C09108=1015.374,-2.873,381.493,-24.167,21.529,-42.895
C09109=1015.372,-2.524,381.465,-24.168,21.529,-42.890
C09110=1015.370,-2.175,381.437,-24.169,21.528,-42.886
C09111=1015.368,-1.829,381.408,-24.169,21.528,-42.880
C09112=1015.365,-1.484,381.381,-24.170,21.527,-42.877
C09113=1015.363,-1.141,381.352,-24.170,21.527,-42.873
C09114=1015.360,-0.799,381.325,-24.171,21.526,-42.867
C09115=1015.359,-0.459,381.298,-24.172,21.526,-42.864
C09116=1015.357,-0.120,381.270,-24.172,21.526,-42.858
C09117=1015.353,0.217,381.242,-24.173,21.525,-42.855
C09118=1015.351,0.553,381.215,-24.173,21.525,-42.851
C09119=1015.350,0.887,381.188,-24.174,21.525,-42.846
C09120=1015.347,1.221,381.161,-24.175,21.524,-42.842
C09121=1015.344,1.555,381.134,-24.175,21.523,-42.838
C09122=1015.342,1.885,381.106,-24.176,21.523,-42.834
C09123=1015.340,2.198,381.082,-24.176,21.523,-42.831
C09124=1015.339,2.486,381.058,-24.177,21.522,-42.827
C09125=1015.336,2.755,381.036,-24.177,21.522,-42.823
C09126=1015.334,3.017,381.015,-24.178,21.522,-42.818
C09127=1015.333,3.286,380.993,-24.179,21.521,-42.814
C09128=1015.330,3.575,380.969,-24.179,21.521,-42.810
C09129=1015.328,3.889,380.943,-24.179,21.520,-42.807
C09130=1015.326,4.218,380.916,-24.180,21.521,-42.803
C09131=1015.323,4.550,380.890,-24.180,21.519,-42.799
C09132=1015.321,4.881,380.862,-24.181,21.519,-42.795
C09133=1015.318,5.211,380.836,-24.181,21.518,-42.792
C09134=1015.316,5.542,380.808,-24.182,21.519,-42.786
C09135=1015.314,5.872,380.782,-24.183,21.518,-42.783
C09136=1015.311,6.201,380.754,-24.183,21.518,-42.779
C09137=1015.308,6.530,380.728,-24.184,21.518,-42.774
C09138=1015.306,6.858,380.701,-24.185,21.517,-42.770
C09139=1015.303,7.186,380.674,-24.185,21.517,-42.766
C09140=1015.301,7.512,380.647,-24.186,21.516,-42.762
C09141=1015.298,7.834,380.620,-24.186,21.516,-42.759
C09142=1015.295,8.155,380.594,-24.186,21.515,-42.755
C09143=1015.294,8.473,380.568,-24.187,21.516,-42.750
C09144=1015.290,8.790,380.542,-24.188,21.515,-42.746
C09145=1015.288,9.105,380.517,-24.188,21.515,-42.742
C09146=1015.285,9.420,380.491,-24.189,21.514,-42.738
C09147=1015.283,9.735,380.465,-24.190,21.514,-42.733
C09148=1015.280,10.050,380.439,-24.190,21.514,-42.730
C09149=1015.278,10.367,380.413,-24.191,21.513,-42.726
C09150=1015.275,10.685,380.387,-24.191,21.513,-42.722
C09151=1015.272,11.006,380.361,-24.192,21.512,-42.718
C09152=1015.269,11.328,380.334,-24.192,21.512,-42.715
C09153=1015.267,11.652,380.307,-24.193,21.511,-42.711
C09154=1015.264,11.975,380.281,-24.193,21.511,-42.707
C09155=1015.261,12.298,380.254,-24.194,21.511,-42.702
C09156=1015.259,12.622,380.227,-24.194,21.510,-42.698
C09157=1015.255,12.945,380.201,-24.195,21.510,-42.694
C09158=1015.253,13.270,380.174,-24.195,21.509,-42.691
C09159=1015.250,13.593,380.148,-24.196,21.509,-42.687
C09160=1015.247,13.918,380.121,-24.197,21.509,-42.682
C09161=1015.244,14.242,380.094,-24.197,21.509,-42.678
C09162=1015.241,14.568,380.068,-24.198,21.508,-42.674
C09163=1015.238,14.893,380.041,-24.198,21.508,-42.670
C09164=1015.235,15.218,380.014,-24.199,21.507,-42.667
C09165=1015.233,15.545,379.987,-24.199,21.507,-42.663
C09166=1015.229,15.872,379.960,-24.200,21.507,-42.658
C09167=1015.227,16.199,379.933,-24.200,21.506,-42.654
C09168=1015.223,16.527,379.906,-24.201,21.506,-42.650
C09169=1015.220,16.856,379.878,-24.201,21.505,-42.646
C09170=1015.217,17.185,379.851,-24.202,21.505,-42.643
C09171=1015.214,17.516,379.824,-24.202,21.504,-42.639
C09172=1015.211,17.845,379.797,-24.203,21.504,-42.634
C09173=1015.208,18.175,379.770,-24.204,21.504,-42.630
C09174=1015.204,18.508,379.742,-24.204,21.503,-42.626
C09175=1015.202,18.839,379.715,-24.205,21.503,-42.622
C09176=1015.198,19.171,379.687,-24.205,21.502,-42.619
C09177=1015.195,19.519,379.658,-24.206,21.503,-42.613
C09178=1015.191,19.937,379.623,-24.207,21.502,-42.608
C09179=1015.188,20.173,379.604,-24.207,21.502,-42.604
C09180=1015.186,20.419,379.584,-24.207,21.502,-42.603
C09181=1015.183,20.668,379.563,-24.208,21.502,-42.601
C09182=1015.180,20.909,379.544,-24.208,21.502,-42.599
C09183=1015.179,21.136,379.524,-24.208,21.501,-42.597
C09184=1015.176,21.344,379.507,-24.209,21.501,-42.593
C09185=1015.172,21.701,379.478,-24.209,21.500,-42.588
C09186=1015.169,22.024,379.451,-24.210,21.501,-42.584
C09187=1015.166,22.319,379.426,-24.210,21.500,-42.582
C09188=1015.164,22.571,379.405,-24.210,21.499,-42.580
C09189=1015.159,22.981,379.371,-24.211,21.499,-42.573
C09190=1015.155,23.388,379.338,-24.212,21.498,-42.565
C09191=1015.153,23.641,379.316,-24.213,21.498,-42.562
C09192=1015.149,23.935,379.292,-24.213,21.498,-42.560
C09193=1015.146,24.262,379.265,-24.213,21.497,-42.558
C09194=1015.143,24.596,379.237,-24.214,21.497,-42.553
C09195=1015.139,24.930,379.209,-24.215,21.497,-42.549
C09196=1015.135,25.264,379.182,-24.215,21.496,-42.545
C09197=1015.132,25.598,379.155,-24.216,21.496,-42.541
C09198=1015.128,25.933,379.127,-24.216,21.495,-42.538
C09199=1015.124,26.266,379.098,-24.217,21.495,-42.534
C09200=1015.121,26.601,379.070,-24.217,21.494,-42.530
C09201=1015.117,26.935,379.043,-24.218,21.494,-42.525
C09202=1015.114,27.269,379.015,-24.219,21.495,-42.522
C09203=1015.110,27.604,378.987,-24.219,21.494,-42.518
C09204=1015.106,27.939,378.959,-24.220,21.494,-42.514
C09205=1015.102,28.273,378.932,-24.220,21.493,-42.510
C09206=1015.098,28.608,378.904,-24.221,21.493,-42.507
C09207=1015.095,28.942,378.876,-24.221,21.492,-42.503
C09208=1015.091,29.276,378.848,-24.222,21.493,-42.498
C09209=1015.087,29.611,378.820,-24.222,21.492,-42.494
C09210=1015.083,29.945,378.792,-24.223,21.492,-42.490
C09211=1015.079,30.280,378.764,-24.223,21.491,-42.486
C09212=1015.075,30.613,378.736,-24.224,21.491,-42.483
C09213=1015.071,30.948,378.708,-24.224,21.490,-42.479
C09214=1015.068,31.282,378.680,-24.225,21.490,-42.475
C09215=1015.063,31.617,378.652,-24.225,21.489,-42.471
C09216=1015.059,31.951,378.624,-24.226,21.489,-42.468
C09217=1015.055,32.286,378.597,-24.226,21.489,-42.464
C09218=1015.051,32.621,378.569,-24.227,21.489,-42.459
C09219=1015.048,32.955,378.541,-24.228,21.489,-42.455
C09220=1015.043,33.290,378.512,-24.228,21.488,-42.452
C09221=1015.039,33.624,378.484,-24.229,21.488,-42.448
C09222=1015.036,33.959,378.456,-24.229,21.487,-42.444
C09223=1015.031,34.294,378.428,-24.230,21.487,-42.440
C09224=1015.027,34.628,378.401,-24.230,21.486,-42.437
C09225=1015.023,34.963,378.373,-24.231,21.486,-42.433
C09226=1015.018,35.297,378.344,-24.231,21.485,-42.429
C09227=1015.014,35.631,378.316,-24.232,21.486,-42.426
C09228=1015.009,35.966,378.289,-24.232,21.485,-42.422
C09229=1015.006,36.301,378.261,-24.233,21.485,-42.418
C09230=1015.001,36.636,378.232,-24.234,21.485,-42.413
C09231=1014.997,36.970,378.204,-24.234,21.485,-42.409
C09232=1014.993,37.305,378.176,-24.235,21.484,-42.405
C09233=1014.989,37.640,378.148,-24.235,21.484,-42.402
C09234=1014.984,37.974,378.120,-24.236,21.483,-42.398
C09235=1014.981,38.309,378.092,-24.236,21.483,-42.395
C09236=1014.976,38.644,378.064,-24.237,21.483,-42.391
C09237=1014.971,38.978,378.036,-24.237,21.483,-42.387
C09238=1014.967,39.313,378.008,-24.238,21.482,-42.383
C09239=1014.962,39.648,377.980,-24.238,21.482,-42.380
C09240=1014.957,39.983,377.952,-24.239,21.481,-42.376
C09241=1014.954,40.317,377.924,-24.239,21.481,-42.372
C09242=1014.949,40.652,377.895,-24.240,21.481,-42.369
C09243=1014.944,40.987,377.867,-24.240,21.481,-42.365
C09244=1014.939,41.321,377.839,-24.241,21.480,-42.361
C09245=1014.935,41.656,377.811,-24.241,21.480,-42.357
C09246=1014.931,41.991,377.783,-24.242,21.479,-42.354
C09247=1014.926,42.326,377.755,-24.242,21.479,-42.350
C09248=1014.921,42.661,377.727,-24.243,21.479,-42.347
C09249=1014.917,42.996,377.698,-24.243,21.479,-42.343
C09250=1014.912,43.330,377.670,-24.244,21.478,-42.339
C09251=1014.907,43.665,377.642,-24.244,21.478,-42.335
C09252=1014.902,44.000,377.614,-24.245,21.477,-42.332
C09253=1014.898,44.335,377.585,-24.245,21.477,-42.328
C09254=1014.893,44.670,377.557,-24.246,21.477,-42.325
C09255=1014.888,45.004,377.529,-24.246,21.477,-42.321
C09256=1014.883,45.339,377.501,-24.247,21.476,-42.317
C09257=1014.879,45.674,377.473,-24.247,21.476,-42.313
C09258=1014.874,46.009,377.445,-24.248,21.475,-42.309
C09259=1014.869,46.343,377.417,-24.248,21.475,-42.306
C09260=1014.864,46.678,377.388,-24.249,21.475,-42.302
C09261=1014.859,47.013,377.361,-24.249,21.475,-42.299
C09262=1014.855,47.348,377.332,-24.250,21.474,-42.295
C09263=1014.849,47.683,377.305,-24.250,21.474,-42.291
C09264=1014.844,48.018,377.275,-24.251,21.473,-42.287
C09265=1014.839,48.353,377.248,-24.251,21.473,-42.284
C09266=1014.834,48.687,377.219,-24.252,21.473,-42.280
C09267=1014.829,49.022,377.192,-24.252,21.473,-42.277
C09268=1014.825,49.357,377.163,-24.253,21.472,-42.273
C09269=1014.819,49.692,377.135,-24.253,21.472,-42.269
C09270=1014.814,50.027,377.106,-24.254,21.472,-42.266
C09271=1014.809,50.362,377.079,-24.254,21.471,-42.262
C09272=1014.803,50.697,377.050,-24.255,21.471,-42.258
C09273=1014.799,51.032,377.022,-24.255,21.471,-42.254
C09274=1014.794,51.367,376.993,-24.256,21.471,-42.251
C09275=1014.788,51.702,376.965,-24.256,21.470,-42.247
C09276=1014.783,52.036,376.937,-24.257,21.470,-42.244
C09277=1014.777,52.371,376.909,-24.257,21.470,-42.240
C09278=1014.773,52.706,376.880,-24.258,21.469,-42.238
C09279=1014.767,53.042,376.852,-24.258,21.469,-42.234
C09280=1014.762,53.376,376.824,-24.259,21.468,-42.230
C09281=1014.757,53.711,376.795,-24.259,21.468,-42.227
C09282=1014.751,54.046,376.768,-24.260,21.468,-42.223
C09283=1014.746,54.381,376.739,-24.260,21.468,-42.220
C09284=1014.740,54.716,376.711,-24.261,21.467,-42.216
C09285=1014.735,55.051,376.682,-24.261,21.467,-42.212
C09286=1014.729,55.386,376.654,-24.262,21.467,-42.209
C09287=1014.724,55.721,376.626,-24.262,21.467,-42.205
C09288=1014.718,56.055,376.597,-24.263,21.466,-42.201
C09289=1014.714,56.391,376.570,-24.263,21.466,-42.197
C09290=1014.708,56.725,376.541,-24.264,21.466,-42.194
C09291=1014.702,57.060,376.513,-24.264,21.465,-42.192
C09292=1014.696,57.396,376.484,-24.264,21.465,-42.188
C09293=1014.691,57.730,376.456,-24.265,21.464,-42.184
C09294=1014.685,58.065,376.428,-24.266,21.465,-42.181
C09295=1014.679,58.400,376.400,-24.266,21.464,-42.177
C09296=1014.673,58.735,376.371,-24.267,21.464,-42.173
C09297=1014.669,59.070,376.343,-24.267,21.464,-42.170
C09298=1014.662,59.405,376.315,-24.268,21.464,-42.166
C09299=1014.656,59.739,376.286,-24.268,21.463,-42.163
C09300=1014.650,60.074,376.258,-24.268,21.462,-42.160
C09301=1014.645,60.410,376.230,-24.269,21.462,-42.157
C09302=1014.639,60.744,376.201,-24.269,21.462,-42.153
C09303=1014.633,61.079,376.173,-24.270,21.461,-42.149
C09304=1014.627,61.414,376.145,-24.270,21.462,-42.146
C09305=1014.622,61.749,376.116,-24.271,21.461,-42.142
C09306=1014.616,62.084,376.088,-24.271,21.461,-42.139
C09307=1014.609,62.420,376.060,-24.272,21.460,-42.135
C09308=1014.603,62.816,376.026,-24.272,21.460,-42.131
C09309=1014.599,63.040,376.007,-24.273,21.461,-42.130
C09310=1014.594,63.258,375.989,-24.273,21.460,-42.128
C09311=1014.589,63.631,375.957,-24.274,21.460,-42.124
C09312=1014.587,63.987,375.923,-24.274,21.459,-42.120
C09313=1014.586,64.373,375.887,-24.274,21.459,-42.116
C09314=1014.584,64.768,375.850,-24.275,21.458,-42.113
C09315=1014.583,65.146,375.815,-24.276,21.459,-42.108
C09316=1014.582,65.500,375.782,-24.276,21.457,-42.105
C09317=1014.581,65.839,375.750,-24.277,21.458,-42.102
C09318=1014.580,66.172,375.719,-24.277,21.457,-42.098
C09319=1014.579,66.508,375.687,-24.278,21.457,-42.094
C09320=1014.578,66.845,375.655,-24.278,21.457,-42.091
C09321=1014.577,67.182,375.623,-24.279,21.457,-42.087
C09322=1014.576,67.520,375.591,-24.279,21.456,-42.085
C09323=1014.575,67.859,375.559,-24.279,21.456,-42.082
C09324=1014.574,68.199,375.527,-24.280,21.456,-42.078
C09325=1014.572,68.541,375.495,-24.280,21.455,-42.074
C09326=1014.571,68.883,375.462,-24.281,21.456,-42.071
C09327=1014.570,69.226,375.431,-24.281,21.455,-42.067
C09328=1014.569,69.570,375.398,-24.282,21.455,-42.063
C09329=1014.568,69.914,375.365,-24.282,21.454,-42.061
C09330=1014.567,70.258,375.333,-24.283,21.454,-42.058
C09331=1014.566,70.604,375.300,-24.283,21.453,-42.054
C09332=1014.564,70.948,375.268,-24.284,21.454,-42.051
C09333=1014.564,71.293,375.235,-24.284,21.453,-42.047
C09334=1014.562,71.637,375.202,-24.285,21.453,-42.043
C09335=1014.560,71.982,375.169,-24.285,21.453,-42.041
C09336=1014.559,72.329,375.136,-24.285,21.452,-42.037
C09337=1014.558,72.676,375.103,-24.286,21.452,-42.034
C09338=1014.558,73.027,375.070,-24.286,21.451,-42.030
C09339=1014.556,73.378,375.037,-24.287,21.452,-42.027
C09340=1014.555,73.731,375.003,-24.288,21.451,-42.023
C09341=1014.554,74.086,374.969,-24.288,21.451,-42.019
C09342=1014.553,74.443,374.935,-24.288,21.451,-42.017
C09343=1014.551,74.801,374.902,-24.289,21.450,-42.013
C09344=1014.550,75.158,374.868,-24.289,21.450,-42.010
C09345=1014.549,75.513,374.834,-24.290,21.450,-42.006
C09346=1014.547,75.861,374.801,-24.290,21.449,-42.004
C09347=1014.546,76.203,374.768,-24.291,21.449,-42.001
C09348=1014.545,76.539,374.736,-24.291,21.449,-41.997
C09349=1014.544,76.869,374.704,-24.292,21.449,-41.994
C09350=1014.543,77.196,374.674,-24.292,21.449,-41.990
C09351=1014.542,77.519,374.643,-24.292,21.448,-41.987
C09352=1014.541,77.843,374.611,-24.293,21.448,-41.984
C09353=1014.539,78.168,374.580,-24.293,21.448,-41.980
C09354=1014.538,78.496,374.549,-24.294,21.447,-41.977
C09355=1014.537,78.828,374.517,-24.295,21.448,-41.973
C09356=1014.536,79.167,374.485,-24.295,21.446,-41.971
C09357=1014.535,79.512,374.452,-24.295,21.447,-41.968
C09358=1014.533,79.863,374.419,-24.296,21.446,-41.964
C09359=1014.532,80.218,374.385,-24.296,21.446,-41.962
C09360=1014.531,80.575,374.351,-24.297,21.446,-41.958
C09361=1014.530,80.931,374.316,-24.297,21.445,-41.955
C09362=1014.528,81.288,374.282,-24.298,21.446,-41.951
C09363=1014.527,81.643,374.248,-24.298,21.445,-41.947
C09364=1014.526,81.997,374.214,-24.298,21.444,-41.945
C09365=1014.524,82.351,374.180,-24.299,21.444,-41.942
C09366=1014.523,82.704,374.146,-24.299,21.444,-41.938
C09367=1014.522,83.056,374.112,-24.300,21.444,-41.935
C09368=1014.520,83.406,374.078,-24.300,21.444,-41.931
C09369=1014.519,83.756,374.045,-24.301,21.443,-41.929
C09370=1014.518,84.106,374.012,-24.301,21.443,-41.925
C09371=1014.517,84.453,373.978,-24.302,21.443,-41.922
C09372=1014.515,84.800,373.944,-24.302,21.443,-41.918
C09373=1014.514,85.145,373.912,-24.302,21.442,-41.916
C09374=1014.513,85.489,373.878,-24.303,21.442,-41.912
C09375=1014.511,85.832,373.845,-24.303,21.442,-41.909
C09376=1014.510,86.175,373.812,-24.304,21.441,-41.906
C09377=1014.509,86.515,373.779,-24.304,21.441,-41.903
C09378=1014.508,86.855,373.746,-24.305,21.441,-41.899
C09379=1014.507,87.192,373.714,-24.305,21.441,-41.898
C09380=1014.505,87.524,373.682,-24.305,21.440,-41.894
C09381=1014.504,87.851,373.649,-24.306,21.441,-41.890
C09382=1014.503,88.173,373.619,-24.306,21.439,-41.888
C09383=1014.502,88.493,373.588,-24.307,21.440,-41.885
C09384=1014.500,88.814,373.557,-24.307,21.439,-41.881
C09385=1014.499,89.138,373.526,-24.308,21.439,-41.879
C09386=1014.498,89.468,373.493,-24.308,21.440,-41.876
C09387=1014.496,89.802,373.461,-24.308,21.438,-41.874
C09388=1014.495,90.136,373.429,-24.309,21.439,-41.870
C09389=1014.494,90.470,373.397,-24.309,21.438,-41.866
C09390=1014.492,90.804,373.364,-24.310,21.438,-41.865
C09391=1014.491,91.139,373.332,-24.310,21.438,-41.861
C09392=1014.490,91.474,373.299,-24.311,21.438,-41.857
C09393=1014.489,91.808,373.266,-24.311,21.437,-41.855
C09394=1014.488,92.142,373.234,-24.311,21.437,-41.852
C09395=1014.486,92.477,373.202,-24.312,21.436,-41.849
C09396=1014.485,92.811,373.169,-24.312,21.437,-41.846
C09397=1014.483,93.145,373.137,-24.313,21.436,-41.842
C09398=1014.482,93.480,373.104,-24.313,21.436,-41.841
C09399=1014.480,93.814,373.072,-24.314,21.436,-41.837
C09400=1014.479,94.148,373.039,-24.314,21.436,-41.833
C09401=1014.478,94.483,373.006,-24.314,21.436,-41.832
C09402=1014.478,94.817,372.974,-24.315,21.435,-41.828
C09403=1014.476,95.151,372.941,-24.315,21.435,-41.826
C09404=1014.475,95.485,372.909,-24.316,21.435,-41.822
C09405=1014.473,95.820,372.876,-24.316,21.435,-41.819
C09406=1014.472,96.154,372.844,-24.316,21.434,-41.817
C09407=1014.470,96.489,372.811,-24.317,21.434,-41.813
C09408=1014.469,96.822,372.778,-24.317,21.434,-41.811
C09409=1014.468,97.157,372.746,-24.318,21.434,-41.808
C09410=1014.466,97.491,372.713,-24.318,21.433,-41.806
C09411=1014.465,97.825,372.681,-24.318,21.433,-41.802
C09412=1014.463,98.159,372.647,-24.319,21.433,-41.799
C09413=1014.462,98.493,372.615,-24.319,21.432,-41.796
C09414=1014.460,98.828,372.582,-24.320,21.433,-41.793
C09415=1014.459,99.162,372.550,-24.320,21.432,-41.791
C09416=1014.458,99.496,372.517,-24.320,21.432,-41.787
C09417=1014.456,99.830,372.484,-24.321,21.432,-41.785
C09418=1014.455,100.164,372.452,-24.321,21.431,-41.782
C09419=1014.454,100.498,372.418,-24.322,21.432,-41.778
C09420=1014.453,100.832,372.387,-24.322,21.431,-41.776
C09421=1014.452,101.166,372.353,-24.323,21.431,-41.773
C09422=1014.450,101.500,372.321,-24.323,21.431,-41.771
C09423=1014.448,101.835,372.288,-24.323,21.430,-41.767
C09424=1014.447,102.169,372.255,-24.324,21.430,-41.765
C09425=1014.445,102.503,372.222,-24.324,21.431,-41.762
C09426=1014.444,102.837,372.189,-24.324,21.429,-41.760
C09427=1014.443,103.171,372.156,-24.325,21.430,-41.756
C09428=1014.441,103.505,372.123,-24.325,21.429,-41.752
C09429=1014.440,103.839,372.091,-24.326,21.429,-41.751
C09430=1014.439,104.173,372.057,-24.326,21.430,-41.747
C09431=1014.437,104.507,372.025,-24.326,21.428,-41.745
C09432=1014.436,104.841,371.992,-24.327,21.429,-41.742
C09433=1014.435,105.175,371.959,-24.327,21.428,-41.739
C09434=1014.433,105.509,371.926,-24.328,21.428,-41.736
C09435=1014.432,105.843,371.893,-24.328,21.428,-41.734
C09436=1014.431,106.177,371.860,-24.328,21.427,-41.730
C09437=1014.429,106.511,371.828,-24.329,21.427,-41.728
C09438=1014.428,106.845,371.794,-24.329,21.428,-41.725
C09439=1014.426,107.180,371.761,-24.329,21.427,-41.723
C09440=1014.425,107.513,371.728,-24.330,21.427,-41.719
C09441=1014.424,107.847,371.695,-24.330,21.427,-41.718
C09442=1014.422,108.182,371.662,-24.331,21.426,-41.714
C09443=1014.421,108.515,371.629,-24.331,21.426,-41.712
C09444=1014.419,108.850,371.597,-24.332,21.426,-41.708
C09445=1014.418,109.183,371.563,-24.332,21.425,-41.706
C09446=1014.416,109.517,371.530,-24.332,21.426,-41.703
C09447=1014.415,109.852,371.497,-24.333,21.425,-41.701
C09448=1014.414,110.185,371.464,-24.333,21.425,-41.697
C09449=1014.412,110.519,371.431,-24.333,21.425,-41.695
C09450=1014.411,110.853,371.398,-24.334,21.424,-41.692
C09451=1014.410,111.187,371.365,-24.334,21.424,-41.690
C09452=1014.408,111.521,371.331,-24.335,21.425,-41.686
C09453=1014.406,111.856,371.299,-24.335,21.423,-41.684
C09454=1014.405,112.189,371.265,-24.335,21.424,-41.681
C09455=1014.404,112.523,371.232,-24.336,21.424,-41.679
C09456=1014.402,112.857,371.198,-24.336,21.423,-41.675
C09457=1014.401,113.191,371.166,-24.336,21.423,-41.673
C09458=1014.399,113.525,371.133,-24.337,21.423,-41.670
C09459=1014.398,113.859,371.099,-24.337,21.422,-41.668
C09460=1014.396,114.193,371.066,-24.338,21.423,-41.664
C09461=1014.395,114.527,371.032,-24.338,21.422,-41.662
C09462=1014.394,114.861,371.000,-24.338,21.421,-41.660
C09463=1014.393,115.195,370.967,-24.339,21.422,-41.657
C09464=1014.391,115.529,370.933,-24.339,21.422,-41.655
C09465=1014.389,115.862,370.900,-24.340,21.422,-41.652
C09466=1014.388,116.196,370.866,-24.340,21.421,-41.649
C09467=1014.386,116.531,370.833,-24.340,21.421,-41.646
C09468=1014.385,116.865,370.800,-24.341,21.421,-41.644
C09469=1014.384,117.198,370.767,-24.341,21.421,-41.640
C09470=1014.382,117.532,370.733,-24.341,21.420,-41.638
C09471=1014.381,117.866,370.700,-24.342,21.421,-41.635
C09472=1014.379,118.200,370.667,-24.342,21.420,-41.633
C09473=1014.378,118.534,370.633,-24.342,21.419,-41.631
C09474=1014.376,118.867,370.600,-24.343,21.420,-41.628
C09475=1014.375,119.202,370.567,-24.343,21.419,-41.625
C09476=1014.373,119.536,370.533,-24.344,21.419,-41.622
C09477=1014.372,119.870,370.500,-24.344,21.419,-41.620
C09478=1014.370,120.204,370.466,-24.345,21.419,-41.617
C09479=1014.369,120.537,370.433,-24.345,21.418,-41.614
C09480=1014.367,120.871,370.400,-24.345,21.418,-41.613
C09481=1014.366,121.205,370.366,-24.346,21.418,-41.609
C09482=1014.364,121.539,370.333,-24.346,21.417,-41.607
C09483=1014.362,121.873,370.299,-24.346,21.418,-41.604
C09484=1014.362,122.207,370.265,-24.347,21.418,-41.602
C09485=1014.360,122.541,370.232,-24.347,21.418,-41.598
C09486=1014.359,122.875,370.198,-24.347,21.417,-41.596
C09487=1014.357,123.209,370.165,-24.348,21.417,-41.594
C09488=1014.356,123.543,370.131,-24.348,21.417,-41.591
C09489=1014.354,123.877,370.098,-24.348,21.417,-41.589
C09490=1014.353,124.210,370.064,-24.349,21.416,-41.585
C09491=1014.351,124.545,370.030,-24.349,21.416,-41.583
C09492=1014.350,124.878,369.997,-24.349,21.416,-41.581
C09493=1014.348,125.213,369.963,-24.350,21.416,-41.578
C09494=1014.347,125.547,369.930,-24.350,21.415,-41.576
C09495=1014.345,125.881,369.896,-24.351,21.416,-41.572
C09496=1014.344,126.214,369.863,-24.351,21.415,-41.571
C09497=1014.342,126.549,369.829,-24.351,21.415,-41.569
C09498=1014.341,126.882,369.796,-24.352,21.415,-41.565
C09499=1014.340,127.217,369.762,-24.352,21.415,-41.563
C09500=1014.338,127.551,369.728,-24.352,21.414,-41.561
C09501=1014.336,127.885,369.695,-24.353,21.415,-41.558
C09502=1014.334,128.219,369.661,-24.353,21.414,-41.555
C09503=1014.333,128.552,369.628,-24.354,21.414,-41.552
C09504=1014.332,128.887,369.593,-24.354,21.414,-41.550
C09505=1014.330,129.221,369.560,-24.354,21.414,-41.548
C09506=1014.329,129.554,369.526,-24.355,21.413,-41.545
C09507=1014.327,129.888,369.492,-24.355,21.413,-41.543
C09508=1014.326,130.223,369.458,-24.355,21.413,-41.541
C09509=1014.325,130.557,369.424,-24.356,21.413,-41.538
C09510=1014.323,130.891,369.391,-24.356,21.412,-41.535
C09511=1014.321,131.225,369.357,-24.356,21.412,-41.532
C09512=1014.320,131.559,369.323,-24.357,21.412,-41.530
C09513=1014.318,131.893,369.289,-24.357,21.412,-41.528
C09514=1014.317,132.227,369.256,-24.357,21.412,-41.525
C09515=1014.316,132.562,369.221,-24.358,21.411,-41.523
C09516=1014.314,132.895,369.187,-24.358,21.411,-41.521
C09517=1014.312,133.229,369.154,-24.358,21.411,-41.517
C09518=1014.311,133.564,369.119,-24.359,21.411,-41.515
C09519=1014.309,133.898,369.086,-24.359,21.410,-41.513
C09520=1014.308,134.232,369.052,-24.359,21.411,-41.510
C09521=1014.307,134.566,369.018,-24.360,21.410,-41.508
C09522=1014.305,134.900,368.984,-24.360,21.410,-41.506
C09523=1014.303,135.234,368.950,-24.361,21.411,-41.503
C09524=1014.302,135.556,368.917,-24.361,21.410,-41.501
C09525=1014.301,135.857,368.886,-24.361,21.410,-41.499
C09526=1014.299,136.136,368.859,-24.361,21.410,-41.497
C09527=1014.298,136.401,368.831,-24.361,21.409,-41.495
C09528=1014.297,136.666,368.804,-24.362,21.409,-41.491
C09529=1014.296,136.941,368.776,-24.362,21.409,-41.490
C09530=1014.294,137.239,368.746,-24.363,21.409,-41.488
C09531=1014.293,137.561,368.713,-24.363,21.408,-41.486
C09532=1014.292,137.901,368.679,-24.363,21.408,-41.484
C09533=1014.290,138.258,368.642,-24.364,21.408,-41.480
C09534=1014.288,138.669,368.600,-24.364,21.408,-41.477
C09535=1014.287,138.897,368.577,-24.364,21.408,-41.475
C09536=1014.286,139.135,368.553,-24.365,21.408,-41.473
C09537=1014.285,139.376,368.528,-24.365,21.408,-41.473
C09538=1014.284,139.617,368.503,-24.365,21.408,-41.471
C09539=1014.283,139.850,368.479,-24.365,21.408,-41.470
C09540=1014.282,140.070,368.457,-24.365,21.407,-41.469
C09541=1014.281,140.463,368.417,-24.366,21.407,-41.465
C09542=1014.279,140.809,368.382,-24.366,21.407,-41.462
C09543=1014.278,141.148,368.347,-24.367,21.407,-41.460
C09544=1014.276,141.487,368.312,-24.367,21.407,-41.457
C09545=1014.274,141.827,368.278,-24.367,21.406,-41.455
C09546=1014.272,142.168,368.242,-24.368,21.406,-41.453
C09547=1014.271,142.509,368.208,-24.368,21.407,-41.449
C09548=1014.270,142.852,368.173,-24.368,21.406,-41.448
C09549=1014.268,143.194,368.137,-24.369,21.405,-41.445
C09550=1014.267,143.537,368.102,-24.369,21.406,-41.442
C09551=1014.264,143.881,368.067,-24.369,21.405,-41.440
C09552=1014.264,144.225,368.032,-24.370,21.405,-41.438
C09553=1014.262,144.569,367.996,-24.370,21.406,-41.435
C09554=1014.261,144.914,367.961,-24.370,21.405,-41.432
C09555=1014.259,145.260,367.925,-24.371,21.404,-41.431
C09556=1014.257,145.605,367.890,-24.371,21.405,-41.427
C09557=1014.255,145.951,367.854,-24.371,21.405,-41.425
C09558=1014.254,146.297,367.819,-24.372,21.404,-41.424
C09559=1014.252,146.644,367.784,-24.372,21.404,-41.420
C09560=1014.248,146.991,367.749,-24.372,21.404,-41.418
C09561=1014.693,147.023,367.472,-24.372,21.404,-41.418
C09562=1014.700,146.676,367.505,-24.372,21.404,-41.420
C09563=1014.701,146.330,367.540,-24.372,21.404,-41.424
C09564=1014.703,145.983,367.576,-24.371,21.405,-41.425
C09565=1014.704,145.638,367.611,-24.371,21.405,-41.427
C09566=1014.706,145.292,367.647,-24.371,21.404,-41.431
C09567=1014.707,144.946,367.682,-24.370,21.405,-41.432
C09568=1014.708,144.602,367.718,-24.370,21.406,-41.435
C09569=1014.710,144.257,367.753,-24.370,21.405,-41.438
C09570=1014.712,143.913,367.788,-24.369,21.405,-41.440
C09571=1014.713,143.570,367.824,-24.369,21.406,-41.442
C09572=1014.715,143.226,367.859,-24.369,21.405,-41.445
C09573=1014.716,142.884,367.894,-24.368,21.406,-41.448
C09574=1014.718,142.542,367.929,-24.368,21.407,-41.449
C09575=1014.719,142.200,367.964,-24.368,21.406,-41.453
C09576=1014.721,141.860,367.999,-24.367,21.406,-41.455
C09577=1014.722,141.520,368.034,-24.367,21.407,-41.457
C09578=1014.724,141.180,368.068,-24.367,21.407,-41.460
C09579=1014.725,140.841,368.103,-24.366,21.407,-41.462
C09580=1014.726,140.496,368.139,-24.366,21.407,-41.465
C09581=1014.728,140.103,368.179,-24.365,21.407,-41.469
C09582=1014.729,139.882,368.201,-24.365,21.408,-41.470
C09583=1014.730,139.649,368.225,-24.365,21.408,-41.471
C09584=1014.732,139.409,368.250,-24.365,21.408,-41.473
C09585=1014.732,139.167,368.275,-24.365,21.408,-41.473
C09586=1014.733,138.929,368.299,-24.364,21.408,-41.475
C09587=1014.734,138.702,368.322,-24.364,21.408,-41.477
C09588=1014.736,138.290,368.364,-24.364,21.408,-41.480
C09589=1014.738,137.933,368.400,-24.363,21.408,-41.484
C09590=1014.739,137.593,368.435,-24.363,21.408,-41.486
C09591=1014.740,137.271,368.468,-24.363,21.409,-41.488
C09592=1014.741,136.974,368.499,-24.362,21.409,-41.490
C09593=1014.743,136.698,368.526,-24.362,21.409,-41.491
C09594=1014.744,136.433,368.553,-24.361,21.409,-41.495
C09595=1014.745,136.168,368.581,-24.361,21.410,-41.497
C09596=1014.746,135.889,368.609,-24.361,21.410,-41.499
C09597=1014.747,135.588,368.640,-24.361,21.410,-41.501
C09598=1014.749,135.266,368.672,-24.361,21.411,-41.503
C09599=1014.751,134.933,368.706,-24.360,21.410,-41.506
C09600=1014.752,134.598,368.740,-24.360,21.410,-41.508
C09601=1014.753,134.264,368.774,-24.359,21.411,-41.510
C09602=1014.755,133.930,368.807,-24.359,21.410,-41.513
C09603=1014.756,133.595,368.842,-24.359,21.411,-41.515
C09604=1014.758,133.262,368.876,-24.358,21.411,-41.517
C09605=1014.759,132.928,368.910,-24.358,21.411,-41.521
C09606=1014.761,132.594,368.944,-24.358,21.411,-41.523
C09607=1014.762,132.260,368.977,-24.357,21.412,-41.525
C09608=1014.764,131.925,369.012,-24.357,21.412,-41.528
C09609=1014.765,131.591,369.045,-24.357,21.412,-41.530
C09610=1014.767,131.258,369.079,-24.356,21.412,-41.532
C09611=1014.768,130.923,369.114,-24.356,21.412,-41.535
C09612=1014.769,130.589,369.147,-24.356,21.413,-41.538
C09613=1014.771,130.255,369.181,-24.355,21.413,-41.541
C09614=1014.773,129.921,369.214,-24.355,21.413,-41.543
C09615=1014.773,129.587,369.248,-24.355,21.413,-41.545
C09616=1014.775,129.253,369.282,-24.354,21.414,-41.548
C09617=1014.777,128.919,369.316,-24.354,21.414,-41.550
C09618=1014.778,128.585,369.350,-24.354,21.414,-41.552
C09619=1014.779,128.251,369.384,-24.353,21.414,-41.555
C09620=1014.781,127.917,369.417,-24.353,21.415,-41.558
C09621=1014.783,127.583,369.451,-24.352,21.414,-41.561
C09622=1014.784,127.249,369.485,-24.352,21.415,-41.563
C09623=1014.785,126.915,369.518,-24.352,21.415,-41.565
C09624=1014.787,126.581,369.552,-24.351,21.415,-41.569
C09625=1014.788,126.247,369.585,-24.351,21.415,-41.571
C09626=1014.790,125.913,369.619,-24.351,21.416,-41.572
C09627=1014.791,125.578,369.653,-24.350,21.415,-41.576
C09628=1014.792,125.245,369.687,-24.350,21.416,-41.578
C09629=1014.793,124.911,369.720,-24.349,21.416,-41.581
C09630=1014.795,124.577,369.754,-24.349,21.416,-41.583
C09631=1014.797,124.243,369.787,-24.349,21.416,-41.585
C09632=1014.798,123.909,369.821,-24.348,21.417,-41.589
C09633=1014.799,123.575,369.855,-24.348,21.417,-41.591
C09634=1014.801,123.241,369.889,-24.348,21.417,-41.594
C09635=1014.802,122.907,369.922,-24.347,21.417,-41.596
C09636=1014.804,122.573,369.956,-24.347,21.418,-41.598
C09637=1014.805,122.239,369.989,-24.347,21.418,-41.602
C09638=1014.807,121.905,370.023,-24.346,21.418,-41.604
C09639=1014.808,121.572,370.056,-24.346,21.417,-41.607
C09640=1014.810,121.238,370.089,-24.346,21.418,-41.609
C09641=1014.811,120.903,370.123,-24.345,21.418,-41.613
C09642=1014.812,120.570,370.156,-24.345,21.418,-41.614
C09643=1014.814,120.236,370.190,-24.345,21.419,-41.617
C09644=1014.815,119.902,370.224,-24.344,21.419,-41.620
C09645=1014.816,119.568,370.257,-24.344,21.419,-41.622
C09646=1014.818,119.234,370.291,-24.343,21.419,-41.625
C09647=1014.820,118.900,370.323,-24.343,21.420,-41.628
C09648=1014.822,118.566,370.357,-24.342,21.419,-41.631
C09649=1014.823,118.232,370.390,-24.342,21.420,-41.633
C09650=1014.824,117.898,370.423,-24.342,21.421,-41.635
C09651=1014.826,117.564,370.457,-24.341,21.420,-41.638
C09652=1014.827,117.230,370.490,-24.341,21.421,-41.640
C09653=1014.828,116.896,370.524,-24.341,21.421,-41.644
C09654=1014.830,116.562,370.558,-24.340,21.421,-41.646
C09655=1014.831,116.228,370.591,-24.340,21.421,-41.649
C09656=1014.832,115.894,370.623,-24.340,21.422,-41.652
C09657=1014.833,115.560,370.657,-24.339,21.422,-41.655
C09658=1014.835,115.226,370.690,-24.339,21.422,-41.657
C09659=1014.836,114.892,370.724,-24.338,21.421,-41.660
C09660=1014.838,114.559,370.757,-24.338,21.422,-41.662
C09661=1014.839,114.225,370.790,-24.338,21.423,-41.664
C09662=1014.841,113.890,370.823,-24.337,21.422,-41.668
C09663=1014.842,113.557,370.856,-24.337,21.423,-41.670
C09664=1014.843,113.223,370.890,-24.336,21.423,-41.673
C09665=1014.845,112.889,370.923,-24.336,21.423,-41.675
C09666=1014.847,112.555,370.957,-24.336,21.424,-41.679
C09667=1014.848,112.221,370.989,-24.335,21.424,-41.681
C09668=1014.849,111.887,371.022,-24.335,21.423,-41.684
C09669=1014.850,111.553,371.056,-24.335,21.425,-41.686
C09670=1014.852,111.220,371.089,-24.334,21.424,-41.690
C09671=1014.854,110.885,371.122,-24.334,21.424,-41.692
C09672=1014.855,110.551,371.155,-24.333,21.425,-41.695
C09673=1014.856,110.218,371.188,-24.333,21.425,-41.697
C09674=1014.858,109.883,371.221,-24.333,21.425,-41.701
C09675=1014.859,109.550,371.254,-24.332,21.426,-41.703
C09676=1014.860,109.216,371.287,-24.332,21.425,-41.706
C09677=1014.862,108.881,371.320,-24.332,21.426,-41.708
C09678=1014.863,108.547,371.354,-24.331,21.426,-41.712
C09679=1014.865,108.214,371.387,-24.331,21.426,-41.714
C09680=1014.866,107.879,371.419,-24.330,21.427,-41.718
C09681=1014.867,107.546,371.453,-24.330,21.427,-41.719
C09682=1014.868,107.212,371.486,-24.329,21.427,-41.723
C09683=1014.870,106.878,371.518,-24.329,21.428,-41.725
C09684=1014.871,106.544,371.552,-24.329,21.427,-41.728
C09685=1014.873,106.210,371.584,-24.328,21.427,-41.730
C09686=1014.874,105.875,371.618,-24.328,21.428,-41.734
C09687=1014.876,105.542,371.651,-24.328,21.428,-41.736
C09688=1014.877,105.207,371.684,-24.327,21.428,-41.739
C09689=1014.878,104.874,371.717,-24.327,21.429,-41.742
C09690=1014.880,104.539,371.749,-24.326,21.428,-41.745
C09691=1014.881,104.206,371.783,-24.326,21.430,-41.747
C09692=1014.882,103.871,371.815,-24.326,21.429,-41.751
C09693=1014.884,103.538,371.848,-24.325,21.429,-41.752
C09694=1014.885,103.203,371.881,-24.325,21.430,-41.756
C09695=1014.886,102.869,371.914,-24.324,21.429,-41.760
C09696=1014.887,102.534,371.947,-24.324,21.431,-41.762
C09697=1014.888,102.201,371.980,-24.324,21.430,-41.765
C09698=1014.890,101.866,372.013,-24.323,21.430,-41.767
C09699=1014.891,101.532,372.045,-24.323,21.431,-41.771
C09700=1014.892,101.198,372.078,-24.323,21.431,-41.773
C09701=1014.894,100.864,372.111,-24.322,21.431,-41.776
C09702=1014.895,100.530,372.144,-24.322,21.432,-41.778
C09703=1014.897,100.196,372.177,-24.321,21.431,-41.782
C09704=1014.898,99.862,372.209,-24.321,21.432,-41.785
C09705=1014.899,99.528,372.242,-24.320,21.432,-41.787
C09706=1014.901,99.193,372.275,-24.320,21.432,-41.791
C09707=1014.902,98.859,372.307,-24.320,21.433,-41.793
C09708=1014.903,98.525,372.340,-24.319,21.432,-41.796
C09709=1014.905,98.191,372.373,-24.319,21.433,-41.799
C09710=1014.906,97.857,372.406,-24.318,21.433,-41.802
C09711=1014.908,97.522,372.438,-24.318,21.433,-41.806
C09712=1014.908,97.189,372.471,-24.318,21.434,-41.808
C09713=1014.910,96.855,372.503,-24.317,21.434,-41.811
C09714=1014.911,96.520,372.536,-24.317,21.434,-41.813
C09715=1014.912,96.186,372.569,-24.316,21.434,-41.817
C09716=1014.913,95.852,372.602,-24.316,21.435,-41.819
C09717=1014.915,95.517,372.634,-24.316,21.435,-41.822
C09718=1014.916,95.183,372.667,-24.315,21.435,-41.826
C09719=1014.918,94.848,372.699,-24.315,21.435,-41.828
C09720=1014.919,94.514,372.732,-24.314,21.436,-41.832
C09721=1014.921,94.180,372.764,-24.314,21.436,-41.833
C09722=1014.921,93.846,372.797,-24.314,21.436,-41.837
C09723=1014.923,93.512,372.829,-24.313,21.436,-41.841
C09724=1014.924,93.177,372.862,-24.313,21.436,-41.842
C09725=1014.925,92.843,372.895,-24.312,21.437,-41.846
C09726=1014.927,92.508,372.927,-24.312,21.436,-41.849
C09727=1014.928,92.174,372.960,-24.311,21.437,-41.852
C09728=1014.930,91.840,372.992,-24.311,21.437,-41.855
C09729=1014.930,91.506,373.024,-24.311,21.438,-41.857
C09730=1014.932,91.171,373.057,-24.310,21.438,-41.861
C09731=1014.933,90.836,373.090,-24.310,21.438,-41.865
C09732=1014.934,90.502,373.122,-24.309,21.438,-41.866
C09733=1014.936,90.167,373.155,-24.309,21.439,-41.870
C09734=1014.937,89.833,373.187,-24.308,21.438,-41.874
C09735=1014.938,89.500,373.219,-24.308,21.440,-41.876
C09736=1014.939,89.170,373.251,-24.308,21.439,-41.879
C09737=1014.940,88.846,373.283,-24.307,21.439,-41.881
C09738=1014.942,88.525,373.314,-24.307,21.440,-41.885
C09739=1014.942,88.204,373.345,-24.306,21.439,-41.888
C09740=1014.943,87.882,373.376,-24.306,21.441,-41.890
C09741=1014.945,87.556,373.407,-24.305,21.440,-41.894
C09742=1014.947,87.224,373.439,-24.305,21.441,-41.898
C09743=1014.948,86.887,373.472,-24.305,21.441,-41.899
C09744=1014.949,86.548,373.505,-24.304,21.441,-41.903
C09745=1014.950,86.206,373.537,-24.304,21.441,-41.906
C09746=1014.951,85.864,373.571,-24.303,21.442,-41.909
C09747=1014.953,85.522,373.604,-24.303,21.442,-41.912
C09748=1014.954,85.177,373.637,-24.302,21.442,-41.916
C09749=1014.955,84.832,373.670,-24.302,21.443,-41.918
C09750=1014.956,84.485,373.704,-24.302,21.443,-41.922
C09751=1014.958,84.137,373.737,-24.301,21.443,-41.925
C09752=1014.959,83.789,373.771,-24.301,21.443,-41.929
C09753=1014.960,83.439,373.804,-24.300,21.444,-41.931
C09754=1014.962,83.087,373.838,-24.300,21.444,-41.935
C09755=1014.962,82.735,373.872,-24.299,21.444,-41.938
C09756=1014.964,82.383,373.906,-24.299,21.444,-41.942
C09757=1014.965,82.029,373.940,-24.298,21.444,-41.945
C09758=1014.967,81.674,373.974,-24.298,21.445,-41.947
C09759=1014.967,81.319,374.008,-24.298,21.446,-41.951
C09760=1014.969,80.963,374.042,-24.297,21.445,-41.955
C09761=1014.971,80.607,374.077,-24.297,21.446,-41.958
C09762=1014.972,80.250,374.111,-24.296,21.446,-41.962
C09763=1014.973,79.895,374.145,-24.296,21.446,-41.964
C09764=1014.974,79.543,374.178,-24.295,21.447,-41.968
C09765=1014.975,79.199,374.211,-24.295,21.446,-41.971
C09766=1014.976,78.860,374.243,-24.295,21.448,-41.973
C09767=1014.977,78.527,374.276,-24.294,21.447,-41.977
C09768=1014.979,78.199,374.307,-24.293,21.448,-41.980
C09769=1014.980,77.874,374.338,-24.293,21.448,-41.984
C09770=1014.981,77.551,374.369,-24.292,21.448,-41.987
C09771=1014.982,77.227,374.400,-24.292,21.449,-41.990
C09772=1014.983,76.901,374.431,-24.292,21.449,-41.994
C09773=1014.984,76.571,374.462,-24.291,21.449,-41.997
C09774=1014.985,76.235,374.495,-24.291,21.449,-42.001
C09775=1014.986,75.893,374.527,-24.290,21.449,-42.004
C09776=1014.988,75.545,374.560,-24.290,21.450,-42.006
C09777=1014.989,75.190,374.594,-24.289,21.450,-42.010
C09778=1014.990,74.833,374.628,-24.289,21.450,-42.013
C09779=1014.992,74.476,374.662,-24.288,21.451,-42.017
C09780=1014.992,74.119,374.696,-24.288,21.451,-42.019
C09781=1014.994,73.762,374.730,-24.288,21.451,-42.023
C09782=1014.995,73.409,374.763,-24.287,21.452,-42.027
C09783=1014.996,73.057,374.797,-24.286,21.451,-42.030
C09784=1014.998,72.708,374.830,-24.286,21.452,-42.034
C09785=1014.998,72.360,374.863,-24.285,21.452,-42.037
C09786=1015.000,72.014,374.896,-24.285,21.453,-42.041
C09787=1015.001,71.669,374.928,-24.285,21.453,-42.043
C09788=1015.002,71.324,374.961,-24.284,21.453,-42.047
C09789=1015.003,70.980,374.994,-24.284,21.454,-42.051
C09790=1015.004,70.635,375.027,-24.283,21.453,-42.054
C09791=1015.005,70.291,375.059,-24.283,21.454,-42.058
C09792=1015.006,69.946,375.092,-24.282,21.454,-42.061
C09793=1015.007,69.602,375.124,-24.282,21.455,-42.063
C09794=1015.008,69.258,375.157,-24.281,21.455,-42.067
C09795=1015.010,68.914,375.190,-24.281,21.456,-42.071
C09796=1015.011,68.572,375.222,-24.280,21.455,-42.074
C09797=1015.012,68.232,375.254,-24.280,21.456,-42.078
C09798=1015.013,67.891,375.286,-24.279,21.456,-42.082
C09799=1015.014,67.552,375.318,-24.279,21.456,-42.085
C09800=1015.015,67.214,375.350,-24.279,21.457,-42.087
C09801=1015.016,66.877,375.382,-24.278,21.457,-42.091
C09802=1015.017,66.540,375.414,-24.278,21.457,-42.094
C09803=1015.018,66.203,375.445,-24.277,21.457,-42.098
C09804=1015.020,65.870,375.477,-24.277,21.458,-42.102
C09805=1015.020,65.532,375.508,-24.276,21.457,-42.105
C09806=1015.022,65.177,375.542,-24.276,21.459,-42.108
C09807=1015.023,64.801,375.577,-24.275,21.458,-42.113
C09808=1015.024,64.405,375.615,-24.274,21.459,-42.116
C09809=1015.025,64.019,375.650,-24.274,21.459,-42.120
C09810=1015.026,63.663,375.684,-24.274,21.460,-42.124
C09811=1015.031,63.289,375.717,-24.273,21.460,-42.128
C09812=1015.035,63.071,375.735,-24.273,21.461,-42.130
C09813=1015.039,62.847,375.754,-24.272,21.460,-42.131
C09814=1015.045,62.451,375.788,-24.272,21.460,-42.135
C09815=1015.051,62.116,375.817,-24.271,21.461,-42.139
C09816=1015.057,61.780,375.845,-24.271,21.461,-42.142
C09817=1015.062,61.446,375.874,-24.270,21.462,-42.146
C09818=1015.067,61.110,375.902,-24.270,21.461,-42.149
C09819=1015.073,60.776,375.931,-24.269,21.462,-42.153
C09820=1015.079,60.440,375.959,-24.269,21.462,-42.157
C09821=1015.085,60.106,375.988,-24.268,21.462,-42.160
C09822=1015.090,59.771,376.017,-24.268,21.463,-42.163
C09823=1015.095,59.436,376.045,-24.268,21.464,-42.166
C09824=1015.100,59.101,376.073,-24.267,21.464,-42.170
C09825=1015.106,58.766,376.102,-24.267,21.464,-42.173
C09826=1015.111,58.431,376.130,-24.266,21.464,-42.177
C09827=1015.117,58.096,376.159,-24.266,21.465,-42.181
C09828=1015.122,57.761,376.188,-24.265,21.464,-42.184
C09829=1015.126,57.426,376.216,-24.264,21.465,-42.188
C09830=1015.133,57.091,376.244,-24.264,21.465,-42.192
C09831=1015.137,56.757,376.273,-24.264,21.466,-42.194
C09832=1015.143,56.421,376.301,-24.263,21.466,-42.197
C09833=1015.149,56.087,376.330,-24.263,21.466,-42.201
C09834=1015.153,55.752,376.359,-24.262,21.467,-42.205
C09835=1015.159,55.416,376.387,-24.262,21.467,-42.209
C09836=1015.163,55.081,376.415,-24.261,21.467,-42.212
C09837=1015.169,54.747,376.444,-24.261,21.467,-42.216
C09838=1015.174,54.412,376.472,-24.260,21.468,-42.220
C09839=1015.178,54.077,376.501,-24.260,21.468,-42.223
C09840=1015.184,53.742,376.530,-24.259,21.468,-42.227
C09841=1015.189,53.407,376.557,-24.259,21.468,-42.230
C09842=1015.194,53.072,376.586,-24.258,21.469,-42.234
C09843=1015.199,52.737,376.614,-24.258,21.469,-42.238
C09844=1015.204,52.402,376.643,-24.257,21.470,-42.240
C09845=1015.209,52.067,376.672,-24.257,21.470,-42.244
C09846=1015.214,51.732,376.700,-24.256,21.470,-42.247
C09847=1015.219,51.398,376.728,-24.256,21.471,-42.251
C09848=1015.224,51.063,376.757,-24.255,21.471,-42.254
C09849=1015.229,50.727,376.785,-24.255,21.471,-42.258
C09850=1015.233,50.393,376.813,-24.254,21.471,-42.262
C09851=1015.238,50.058,376.842,-24.254,21.472,-42.266
C09852=1015.243,49.723,376.871,-24.253,21.472,-42.269
C09853=1015.248,49.388,376.899,-24.253,21.472,-42.273
C09854=1015.252,49.053,376.927,-24.252,21.473,-42.277
C09855=1015.257,48.718,376.956,-24.252,21.473,-42.280
C09856=1015.262,48.384,376.983,-24.251,21.473,-42.284
C09857=1015.267,48.049,377.012,-24.251,21.473,-42.287
C09858=1015.272,47.714,377.041,-24.250,21.474,-42.291
C09859=1015.277,47.379,377.070,-24.250,21.474,-42.295
C09860=1015.281,47.044,377.097,-24.249,21.475,-42.299
C09861=1015.286,46.709,377.126,-24.249,21.475,-42.302
C09862=1015.291,46.374,377.155,-24.248,21.475,-42.306
C09863=1015.295,46.039,377.182,-24.248,21.475,-42.309
C09864=1015.300,45.704,377.211,-24.247,21.476,-42.313
C09865=1015.304,45.370,377.239,-24.247,21.476,-42.317
C09866=1015.308,45.108,377.262,-24.246,21.476,-42.319
C09867=1015.314,44.699,377.296,-24.246,21.477,-42.325
C09868=1015.317,44.365,377.324,-24.245,21.477,-42.328
C09869=1015.322,44.030,377.352,-24.245,21.477,-42.332
C09870=1015.326,43.696,377.381,-24.244,21.478,-42.335
C09871=1015.331,43.361,377.409,-24.244,21.478,-42.339
C09872=1015.336,43.026,377.437,-24.243,21.479,-42.343
C09873=1015.340,42.691,377.466,-24.243,21.479,-42.347
C09874=1015.344,42.356,377.494,-24.242,21.479,-42.350
C09875=1015.349,42.022,377.522,-24.242,21.479,-42.354
C09876=1015.353,41.687,377.551,-24.241,21.480,-42.357
C09877=1015.358,41.352,377.579,-24.241,21.480,-42.361
C09878=1015.361,41.016,377.607,-24.240,21.481,-42.365
C09879=1015.366,40.682,377.636,-24.240,21.481,-42.369
C09880=1015.370,40.347,377.664,-24.239,21.481,-42.372
C09881=1015.374,40.013,377.692,-24.239,21.481,-42.376
C09882=1015.378,39.678,377.721,-24.238,21.482,-42.380
C09883=1015.383,39.343,377.748,-24.238,21.482,-42.383
C09884=1015.387,39.008,377.776,-24.237,21.483,-42.387
C09885=1015.392,38.673,377.805,-24.237,21.483,-42.391
C09886=1015.395,38.339,377.833,-24.236,21.483,-42.395
C09887=1015.400,38.004,377.861,-24.236,21.483,-42.398
C09888=1015.404,37.670,377.889,-24.235,21.484,-42.402
C09889=1015.408,37.335,377.918,-24.235,21.484,-42.405
C09890=1015.412,37.001,377.946,-24.234,21.485,-42.409
C09891=1015.416,36.666,377.974,-24.234,21.485,-42.413
C09892=1015.420,36.330,378.002,-24.233,21.485,-42.418
C09893=1015.424,35.996,378.030,-24.232,21.485,-42.422
C09894=1015.428,35.661,378.058,-24.232,21.486,-42.426
C09895=1015.432,35.327,378.086,-24.231,21.485,-42.429
C09896=1015.436,34.992,378.114,-24.231,21.486,-42.433
C09897=1015.440,34.658,378.143,-24.230,21.486,-42.437
C09898=1015.444,34.323,378.171,-24.230,21.487,-42.440
C09899=1015.448,33.989,378.199,-24.229,21.487,-42.444
C09900=1015.452,33.654,378.227,-24.229,21.488,-42.448
C09901=1015.456,33.320,378.255,-24.228,21.488,-42.452
C09902=1015.459,32.985,378.284,-24.228,21.489,-42.455
C09903=1015.463,32.650,378.312,-24.227,21.489,-42.459
C09904=1015.467,32.316,378.339,-24.226,21.489,-42.464
C09905=1015.471,31.981,378.367,-24.226,21.489,-42.468
C09906=1015.475,31.647,378.396,-24.225,21.489,-42.471
C09907=1015.479,31.312,378.424,-24.225,21.490,-42.475
C09908=1015.483,30.978,378.452,-24.224,21.490,-42.479
C09909=1015.486,30.643,378.480,-24.224,21.491,-42.483
C09910=1015.490,30.309,378.508,-24.223,21.491,-42.486
C09911=1015.493,29.974,378.536,-24.223,21.492,-42.490
C09912=1015.497,29.640,378.564,-24.222,21.492,-42.494
C09913=1015.501,29.305,378.592,-24.222,21.493,-42.498
C09914=1015.505,28.971,378.620,-24.221,21.492,-42.503
C09915=1015.508,28.636,378.648,-24.221,21.493,-42.507
C09916=1015.512,28.303,378.677,-24.220,21.493,-42.510
C09917=1015.515,27.968,378.704,-24.220,21.494,-42.514
C09918=1015.519,27.634,378.732,-24.219,21.494,-42.518
C09919=1015.523,27.300,378.760,-24.219,21.495,-42.522
C09920=1015.526,26.965,378.788,-24.218,21.494,-42.525
C09921=1015.530,26.631,378.816,-24.217,21.494,-42.530
C09922=1015.533,26.296,378.843,-24.217,21.495,-42.534
C09923=1015.536,25.962,378.871,-24.216,21.495,-42.538
C09924=1015.540,25.627,378.899,-24.216,21.496,-42.541
C09925=1015.543,25.294,378.927,-24.215,21.496,-42.545
C09926=1015.547,24.959,378.955,-24.215,21.497,-42.549
C09927=1015.550,24.625,378.983,-24.214,21.497,-42.553
C09928=1015.553,24.291,379.011,-24.213,21.497,-42.558
C09929=1015.556,23.964,379.039,-24.213,21.498,-42.560
C09930=1015.560,23.670,379.062,-24.213,21.498,-42.562
C09931=1015.562,23.418,379.084,-24.212,21.498,-42.565
C09932=1015.567,23.010,379.118,-24.211,21.499,-42.573
C09933=1015.570,22.600,379.152,-24.210,21.499,-42.580
C09934=1015.573,22.348,379.173,-24.210,21.500,-42.582
C09935=1015.575,22.053,379.198,-24.210,21.501,-42.584
C09936=1015.579,21.730,379.225,-24.209,21.500,-42.588
C09937=1015.583,21.372,379.254,-24.209,21.501,-42.593
C09938=1015.585,21.166,379.271,-24.208,21.501,-42.597
C09939=1015.586,20.938,379.290,-24.208,21.502,-42.599
C09940=1015.589,20.697,379.310,-24.208,21.502,-42.601
C09941=1015.591,20.448,379.331,-24.207,21.502,-42.603
C09942=1015.594,20.202,379.352,-24.207,21.502,-42.604
C09943=1015.596,19.966,379.371,-24.207,21.502,-42.608
C09944=1015.600,19.548,379.406,-24.206,21.503,-42.613
C09945=1015.603,19.200,379.435,-24.205,21.502,-42.619
C09946=1015.607,18.868,379.462,-24.205,21.503,-42.622
C09947=1015.609,18.537,379.490,-24.204,21.503,-42.626
C09948=1015.612,18.206,379.517,-24.204,21.504,-42.630
C09949=1015.615,17.875,379.544,-24.203,21.504,-42.634
C09950=1015.618,17.544,379.572,-24.202,21.504,-42.639
C09951=1015.621,17.214,379.600,-24.202,21.505,-42.643
C09952=1015.624,16.886,379.626,-24.201,21.505,-42.646
C09953=1015.627,16.557,379.653,-24.201,21.506,-42.650
C09954=1015.630,16.229,379.681,-24.200,21.506,-42.654
C09955=1015.633,15.901,379.708,-24.200,21.507,-42.658
C09956=1015.636,15.574,379.735,-24.199,21.507,-42.663
C09957=1015.638,15.248,379.762,-24.199,21.507,-42.667
C09958=1015.642,14.922,379.789,-24.198,21.508,-42.670
C09959=1015.644,14.596,379.816,-24.198,21.508,-42.674
C09960=1015.648,14.271,379.842,-24.197,21.509,-42.678
C09961=1015.650,13.946,379.870,-24.197,21.509,-42.682
C09962=1015.653,13.622,379.897,-24.196,21.509,-42.687
C09963=1015.656,13.299,379.923,-24.195,21.509,-42.691
C09964=1015.658,12.975,379.950,-24.195,21.510,-42.694
C09965=1015.660,12.651,379.977,-24.194,21.510,-42.698
C09966=1015.663,12.327,380.003,-24.194,21.511,-42.702
C09967=1015.666,12.004,380.030,-24.193,21.511,-42.707
C09968=1015.669,11.680,380.057,-24.193,21.511,-42.711
C09969=1015.672,11.357,380.083,-24.192,21.512,-42.715
C09970=1015.674,11.035,380.111,-24.192,21.512,-42.718
C09971=1015.676,10.714,380.136,-24.191,21.513,-42.722
C09972=1015.680,10.395,380.163,-24.191,21.513,-42.726
C09973=1015.682,10.079,380.188,-24.190,21.514,-42.730
C09974=1015.684,9.763,380.214,-24.190,21.514,-42.733
C09975=1015.687,9.448,380.240,-24.189,21.514,-42.738
C09976=1015.689,9.134,380.266,-24.188,21.515,-42.742
C09977=1015.692,8.819,380.292,-24.188,21.515,-42.746
C09978=1015.694,8.502,380.318,-24.187,21.516,-42.750
C09979=1015.697,8.184,380.344,-24.186,21.515,-42.755
C09980=1015.699,7.863,380.371,-24.186,21.516,-42.759
C09981=1015.701,7.540,380.397,-24.186,21.516,-42.762
C09982=1015.704,7.215,380.424,-24.185,21.517,-42.766
C09983=1015.707,6.888,380.451,-24.185,21.517,-42.770
C09984=1015.708,6.559,380.478,-24.184,21.518,-42.774
C09985=1015.711,6.230,380.505,-24.183,21.518,-42.779
C09986=1015.714,5.900,380.532,-24.183,21.518,-42.783
//INST
///DATE 2021/06/25 14:57
///ATTR SC,RW,RJ
////FRAME USER -1
///GROUP1 RB1
NOP
MOVJ C00000 VJ=100.00 PL=0
MOVJ C00001 VJ=100.00 PL=0
'Path Start: Op_ID_1
MOVJ C00002 VJ=25.00 PL=0
MOVJ C00003 VJ=25.00 PL=0
'CALL JOB: TOOL ON
MOVL C00004 V=800.0 PL=0
MOVL C00005 V=800.0 PL=0
MOVL C00006 V=800.0 PL=0
MOVL C00007 V=800.0 PL=0
MOVL C00008 V=800.0 PL=0
MOVL C00009 V=800.0 PL=0
MOVL C00010 V=800.0 PL=0
MOVL C00011 V=800.0 PL=0
MOVL C00012 V=800.0 PL=0
MOVL C00013 V=800.0 PL=0
MOVL C00014 V=800.0 PL=0
MOVL C00015 V=800.0 PL=0
MOVL C00016 V=800.0 PL=0
MOVL C00017 V=800.0 PL=0
MOVL C00018 V=800.0 PL=0
MOVL C00019 V=800.0 PL=0
MOVL C00020 V=800.0 PL=0
MOVL C00021 V=800.0 PL=0
MOVL C00022 V=800.0 PL=0
MOVL C00023 V=800.0 PL=0
MOVL C00024 V=800.0 PL=0
MOVL C00025 V=800.0 PL=0
MOVL C00026 V=800.0 PL=0
MOVL C00027 V=800.0 PL=0
MOVL C00028 V=800.0 PL=0
MOVL C00029 V=800.0 PL=0
MOVL C00030 V=800.0 PL=0
MOVL C00031 V=800.0 PL=0
MOVL C00032 V=800.0 PL=0
MOVL C00033 V=800.0 PL=0
MOVL C00034 V=800.0 PL=0
MOVL C00035 V=800.0 PL=0
MOVL C00036 V=800.0 PL=0
MOVL C00037 V=800.0 PL=0
MOVL C00038 V=800.0 PL=0
MOVL C00039 V=800.0 PL=0
MOVL C00040 V=800.0 PL=0
MOVL C00041 V=800.0 PL=0
MOVL C00042 V=800.0 PL=0
MOVL C00043 V=800.0 PL=0
MOVL C00044 V=800.0 PL=0
MOVL C00045 V=800.0 PL=0
MOVL C00046 V=800.0 PL=0
MOVL C00047 V=800.0 PL=0
MOVL C00048 V=800.0 PL=0
MOVL C00049 V=800.0 PL=0
MOVL C00050 V=800.0 PL=0
MOVL C00051 V=800.0 PL=0
MOVL C00052 V=800.0 PL=0
MOVL C00053 V=800.0 PL=0
MOVL C00054 V=800.0 PL=0
MOVL C00055 V=800.0 PL=0
MOVL C00056 V=800.0 PL=0
MOVL C00057 V=800.0 PL=0
MOVL C00058 V=800.0 PL=0
MOVL C00059 V=800.0 PL=0
MOVL C00060 V=800.0 PL=0
MOVL C00061 V=800.0 PL=0
MOVL C00062 V=800.0 PL=0
MOVL C00063 V=800.0 PL=0
MOVL C00064 V=800.0 PL=0
MOVL C00065 V=800.0 PL=0
MOVL C00066 V=800.0 PL=0
MOVL C00067 V=800.0 PL=0
MOVL C00068 V=800.0 PL=0
MOVL C00069 V=800.0 PL=0
MOVL C00070 V=800.0 PL=0
MOVL C00071 V=800.0 PL=0
MOVL C00072 V=800.0 PL=0
MOVL C00073 V=800.0 PL=0
MOVL C00074 V=800.0 PL=0
MOVL C00075 V=800.0 PL=0
MOVL C00076 V=800.0 PL=0
MOVL C00077 V=800.0 PL=0
MOVL C00078 V=800.0 PL=0
MOVL C00079 V=800.0 PL=0
MOVL C00080 V=800.0 PL=0
MOVL C00081 V=800.0 PL=0
MOVL C00082 V=800.0 PL=0
MOVL C00083 V=800.0 PL=0
MOVL C00084 V=800.0 PL=0
MOVL C00085 V=800.0 PL=0
MOVL C00086 V=800.0 PL=0
MOVL C00087 V=800.0 PL=0
MOVL C00088 V=800.0 PL=0
MOVL C00089 V=800.0 PL=0
MOVL C00090 V=800.0 PL=0
MOVL C00091 V=800.0 PL=0
MOVL C00092 V=800.0 PL=0
MOVL C00093 V=800.0 PL=0
MOVL C00094 V=800.0 PL=0
MOVL C00095 V=800.0 PL=0
MOVL C00096 V=800.0 PL=0
MOVL C00097 V=800.0 PL=0
MOVL C00098 V=800.0 PL=0
MOVL C00099 V=800.0 PL=0
MOVL C00100 V=800.0 PL=0
MOVL C00101 V=800.0 PL=0
MOVL C00102 V=800.0 PL=0
MOVL C00103 V=800.0 PL=0
MOVL C00104 V=800.0 PL=0
MOVL C00105 V=800.0 PL=0
MOVL C00106 V=800.0 PL=0
MOVL C00107 V=800.0 PL=0
MOVL C00108 V=800.0 PL=0
MOVL C00109 V=800.0 PL=0
MOVL C00110 V=800.0 PL=0
MOVL C00111 V=800.0 PL=0
MOVL C00112 V=800.0 PL=0
MOVL C00113 V=800.0 PL=0
MOVL C00114 V=800.0 PL=0
MOVL C00115 V=800.0 PL=0
MOVL C00116 V=800.0 PL=0
MOVL C00117 V=800.0 PL=0
MOVL C00118 V=800.0 PL=0
MOVL C00119 V=800.0 PL=0
MOVL C00120 V=800.0 PL=0
MOVL C00121 V=800.0 PL=0
MOVL C00122 V=800.0 PL=0
MOVL C00123 V=800.0 PL=0
MOVL C00124 V=800.0 PL=0
MOVL C00125 V=800.0 PL=0
MOVL C00126 V=800.0 PL=0
MOVL C00127 V=800.0 PL=0
MOVL C00128 V=800.0 PL=0
MOVL C00129 V=800.0 PL=0
MOVL C00130 V=800.0 PL=0
MOVL C00131 V=800.0 PL=0
MOVL C00132 V=800.0 PL=0
MOVL C00133 V=800.0 PL=0
MOVL C00134 V=800.0 PL=0
MOVL C00135 V=800.0 PL=0
MOVL C00136 V=800.0 PL=0
MOVL C00137 V=800.0 PL=0
MOVL C00138 V=800.0 PL=0
MOVL C00139 V=800.0 PL=0
MOVL C00140 V=800.0 PL=0
MOVL C00141 V=800.0 PL=0
MOVL C00142 V=800.0 PL=0
MOVL C00143 V=800.0 PL=0
MOVL C00144 V=800.0 PL=0
MOVL C00145 V=800.0 PL=0
MOVL C00146 V=800.0 PL=0
MOVL C00147 V=800.0 PL=0
MOVL C00148 V=800.0 PL=0
MOVL C00149 V=800.0 PL=0
MOVL C00150 V=800.0 PL=0
MOVL C00151 V=800.0 PL=0
MOVL C00152 V=800.0 PL=0
MOVL C00153 V=800.0 PL=0
MOVL C00154 V=800.0 PL=0
MOVL C00155 V=800.0 PL=0
MOVL C00156 V=800.0 PL=0
MOVL C00157 V=800.0 PL=0
MOVL C00158 V=800.0 PL=0
MOVL C00159 V=800.0 PL=0
MOVL C00160 V=800.0 PL=0
MOVL C00161 V=800.0 PL=0
MOVL C00162 V=800.0 PL=0
MOVL C00163 V=800.0 PL=0
MOVL C00164 V=800.0 PL=0
MOVL C00165 V=800.0 PL=0
MOVL C00166 V=800.0 PL=0
MOVL C00167 V=800.0 PL=0
MOVL C00168 V=800.0 PL=0
MOVL C00169 V=800.0 PL=0
MOVL C00170 V=800.0 PL=0
MOVL C00171 V=800.0 PL=0
MOVL C00172 V=800.0 PL=0
MOVL C00173 V=800.0 PL=0
MOVL C00174 V=800.0 PL=0
MOVL C00175 V=800.0 PL=0
MOVL C00176 V=800.0 PL=0
MOVL C00177 V=800.0 PL=0
MOVL C00178 V=800.0 PL=0
MOVL C00179 V=800.0 PL=0
MOVL C00180 V=800.0 PL=0
MOVL C00181 V=800.0 PL=0
MOVL C00182 V=800.0 PL=0
MOVL C00183 V=800.0 PL=0
MOVL C00184 V=800.0 PL=0
MOVL C00185 V=800.0 PL=0
MOVL C00186 V=800.0 PL=0
MOVL C00187 V=800.0 PL=0
MOVL C00188 V=800.0 PL=0
MOVL C00189 V=800.0 PL=0
MOVL C00190 V=800.0 PL=0
MOVL C00191 V=800.0 PL=0
MOVL C00192 V=800.0 PL=0
MOVL C00193 V=800.0 PL=0
MOVL C00194 V=800.0 PL=0
MOVL C00195 V=800.0 PL=0
MOVL C00196 V=800.0 PL=0
MOVL C00197 V=800.0 PL=0
MOVL C00198 V=800.0 PL=0
MOVL C00199 V=800.0 PL=0
MOVL C00200 V=800.0 PL=0
MOVL C00201 V=800.0 PL=0
MOVL C00202 V=800.0 PL=0
MOVL C00203 V=800.0 PL=0
MOVL C00204 V=800.0 PL=0
MOVL C00205 V=800.0 PL=0
MOVL C00206 V=800.0 PL=0
MOVL C00207 V=800.0 PL=0
MOVL C00208 V=800.0 PL=0
MOVL C00209 V=800.0 PL=0
MOVL C00210 V=800.0 PL=0
MOVL C00211 V=800.0 PL=0
MOVL C00212 V=800.0 PL=0
MOVL C00213 V=800.0 PL=0
MOVL C00214 V=800.0 PL=0
MOVL C00215 V=800.0 PL=0
MOVL C00216 V=800.0 PL=0
MOVL C00217 V=800.0 PL=0
MOVL C00218 V=800.0 PL=0
MOVL C00219 V=800.0 PL=0
MOVL C00220 V=800.0 PL=0
MOVL C00221 V=800.0 PL=0
MOVL C00222 V=800.0 PL=0
MOVL C00223 V=800.0 PL=0
MOVL C00224 V=800.0 PL=0
MOVL C00225 V=800.0 PL=0
MOVL C00226 V=800.0 PL=0
MOVL C00227 V=800.0 PL=0
MOVL C00228 V=800.0 PL=0
MOVL C00229 V=800.0 PL=0
MOVL C00230 V=800.0 PL=0
MOVL C00231 V=800.0 PL=0
MOVL C00232 V=800.0 PL=0
MOVL C00233 V=800.0 PL=0
MOVL C00234 V=800.0 PL=0
MOVL C00235 V=800.0 PL=0
MOVL C00236 V=800.0 PL=0
MOVL C00237 V=800.0 PL=0
MOVL C00238 V=800.0 PL=0
MOVL C00239 V=800.0 PL=0
MOVL C00240 V=800.0 PL=0
MOVL C00241 V=800.0 PL=0
MOVL C00242 V=800.0 PL=0
MOVL C00243 V=800.0 PL=0
MOVL C00244 V=800.0 PL=0
MOVL C00245 V=800.0 PL=0
MOVL C00246 V=800.0 PL=0
MOVL C00247 V=800.0 PL=0
MOVL C00248 V=800.0 PL=0
MOVL C00249 V=800.0 PL=0
MOVL C00250 V=800.0 PL=0
MOVL C00251 V=800.0 PL=0
MOVL C00252 V=800.0 PL=0
MOVL C00253 V=800.0 PL=0
MOVL C00254 V=800.0 PL=0
MOVL C00255 V=800.0 PL=0
MOVL C00256 V=800.0 PL=0
MOVL C00257 V=800.0 PL=0
MOVL C00258 V=800.0 PL=0
MOVL C00259 V=800.0 PL=0
MOVL C00260 V=800.0 PL=0
MOVL C00261 V=800.0 PL=0
MOVL C00262 V=800.0 PL=0
MOVL C00263 V=800.0 PL=0
MOVL C00264 V=800.0 PL=0
MOVL C00265 V=800.0 PL=0
MOVL C00266 V=800.0 PL=0
MOVL C00267 V=800.0 PL=0
MOVL C00268 V=800.0 PL=0
MOVL C00269 V=800.0 PL=0
MOVL C00270 V=800.0 PL=0
MOVL C00271 V=800.0 PL=0
MOVL C00272 V=800.0 PL=0
MOVL C00273 V=800.0 PL=0
MOVL C00274 V=800.0 PL=0
MOVL C00275 V=800.0 PL=0
MOVL C00276 V=800.0 PL=0
MOVL C00277 V=800.0 PL=0
MOVL C00278 V=800.0 PL=0
MOVL C00279 V=800.0 PL=0
MOVL C00280 V=800.0 PL=0
MOVL C00281 V=800.0 PL=0
MOVL C00282 V=800.0 PL=0
MOVL C00283 V=800.0 PL=0
MOVL C00284 V=800.0 PL=0
MOVL C00285 V=800.0 PL=0
MOVL C00286 V=800.0 PL=0
MOVL C00287 V=800.0 PL=0
MOVL C00288 V=800.0 PL=0
MOVL C00289 V=800.0 PL=0
MOVL C00290 V=800.0 PL=0
MOVL C00291 V=800.0 PL=0
MOVL C00292 V=800.0 PL=0
MOVL C00293 V=800.0 PL=0
MOVL C00294 V=800.0 PL=0
MOVL C00295 V=800.0 PL=0
MOVL C00296 V=800.0 PL=0
MOVL C00297 V=800.0 PL=0
MOVL C00298 V=800.0 PL=0
MOVL C00299 V=800.0 PL=0
MOVL C00300 V=800.0 PL=0
MOVL C00301 V=800.0 PL=0
MOVL C00302 V=800.0 PL=0
MOVL C00303 V=800.0 PL=0
MOVL C00304 V=800.0 PL=0
MOVL C00305 V=800.0 PL=0
MOVL C00306 V=800.0 PL=0
MOVL C00307 V=800.0 PL=0
MOVL C00308 V=800.0 PL=0
MOVL C00309 V=800.0 PL=0
MOVL C00310 V=800.0 PL=0
MOVL C00311 V=800.0 PL=0
MOVL C00312 V=800.0 PL=0
MOVL C00313 V=800.0 PL=0
MOVL C00314 V=800.0 PL=0
MOVL C00315 V=800.0 PL=0
MOVL C00316 V=800.0 PL=0
MOVL C00317 V=800.0 PL=0
MOVL C00318 V=800.0 PL=0
MOVL C00319 V=800.0 PL=0
MOVL C00320 V=800.0 PL=0
MOVL C00321 V=800.0 PL=0
MOVL C00322 V=800.0 PL=0
MOVL C00323 V=800.0 PL=0
MOVL C00324 V=800.0 PL=0
MOVL C00325 V=800.0 PL=0
MOVL C00326 V=800.0 PL=0
MOVL C00327 V=800.0 PL=0
MOVL C00328 V=800.0 PL=0
MOVL C00329 V=800.0 PL=0
MOVL C00330 V=800.0 PL=0
MOVL C00331 V=800.0 PL=0
MOVL C00332 V=800.0 PL=0
MOVL C00333 V=800.0 PL=0
MOVL C00334 V=800.0 PL=0
MOVL C00335 V=800.0 PL=0
MOVL C00336 V=800.0 PL=0
MOVL C00337 V=800.0 PL=0
MOVL C00338 V=800.0 PL=0
MOVL C00339 V=800.0 PL=0
MOVL C00340 V=800.0 PL=0
MOVL C00341 V=800.0 PL=0
MOVL C00342 V=800.0 PL=0
MOVL C00343 V=800.0 PL=0
MOVL C00344 V=800.0 PL=0
MOVL C00345 V=800.0 PL=0
MOVL C00346 V=800.0 PL=0
MOVL C00347 V=800.0 PL=0
MOVL C00348 V=800.0 PL=0
MOVL C00349 V=800.0 PL=0
MOVL C00350 V=800.0 PL=0
MOVL C00351 V=800.0 PL=0
MOVL C00352 V=800.0 PL=0
MOVL C00353 V=800.0 PL=0
MOVL C00354 V=800.0 PL=0
MOVL C00355 V=800.0 PL=0
MOVL C00356 V=800.0 PL=0
MOVL C00357 V=800.0 PL=0
MOVL C00358 V=800.0 PL=0
MOVL C00359 V=800.0 PL=0
MOVL C00360 V=800.0 PL=0
MOVL C00361 V=800.0 PL=0
MOVL C00362 V=800.0 PL=0
MOVL C00363 V=800.0 PL=0
MOVL C00364 V=800.0 PL=0
MOVL C00365 V=800.0 PL=0
MOVL C00366 V=800.0 PL=0
MOVL C00367 V=800.0 PL=0
MOVL C00368 V=800.0 PL=0
MOVL C00369 V=800.0 PL=0
MOVL C00370 V=800.0 PL=0
MOVL C00371 V=800.0 PL=0
MOVL C00372 V=800.0 PL=0
MOVL C00373 V=800.0 PL=0
MOVL C00374 V=800.0 PL=0
MOVL C00375 V=800.0 PL=0
MOVL C00376 V=800.0 PL=0
MOVL C00377 V=800.0 PL=0
MOVL C00378 V=800.0 PL=0
MOVL C00379 V=800.0 PL=0
MOVL C00380 V=800.0 PL=0
MOVL C00381 V=800.0 PL=0
MOVL C00382 V=800.0 PL=0
MOVL C00383 V=800.0 PL=0
MOVL C00384 V=800.0 PL=0
MOVL C00385 V=800.0 PL=0
MOVL C00386 V=800.0 PL=0
MOVL C00387 V=800.0 PL=0
MOVL C00388 V=800.0 PL=0
MOVL C00389 V=800.0 PL=0
MOVL C00390 V=800.0 PL=0
'CALL JOB: TOOL OFF
MOVJ C00391 VJ=25.00 PL=0
'CALL JOB: TOOL ON
MOVL C00392 V=800.0 PL=0
MOVL C00393 V=800.0 PL=0
MOVL C00394 V=800.0 PL=0
MOVL C00395 V=800.0 PL=0
MOVL C00396 V=800.0 PL=0
MOVL C00397 V=800.0 PL=0
MOVL C00398 V=800.0 PL=0
MOVL C00399 V=800.0 PL=0
MOVL C00400 V=800.0 PL=0
MOVL C00401 V=800.0 PL=0
MOVL C00402 V=800.0 PL=0
MOVL C00403 V=800.0 PL=0
MOVL C00404 V=800.0 PL=0
MOVL C00405 V=800.0 PL=0
MOVL C00406 V=800.0 PL=0
MOVL C00407 V=800.0 PL=0
MOVL C00408 V=800.0 PL=0
MOVL C00409 V=800.0 PL=0
MOVL C00410 V=800.0 PL=0
MOVL C00411 V=800.0 PL=0
MOVL C00412 V=800.0 PL=0
MOVL C00413 V=800.0 PL=0
MOVL C00414 V=800.0 PL=0
MOVL C00415 V=800.0 PL=0
MOVL C00416 V=800.0 PL=0
MOVL C00417 V=800.0 PL=0
MOVL C00418 V=800.0 PL=0
MOVL C00419 V=800.0 PL=0
MOVL C00420 V=800.0 PL=0
MOVL C00421 V=800.0 PL=0
MOVL C00422 V=800.0 PL=0
MOVL C00423 V=800.0 PL=0
MOVL C00424 V=800.0 PL=0
MOVL C00425 V=800.0 PL=0
MOVL C00426 V=800.0 PL=0
MOVL C00427 V=800.0 PL=0
MOVL C00428 V=800.0 PL=0
MOVL C00429 V=800.0 PL=0
MOVL C00430 V=800.0 PL=0
MOVL C00431 V=800.0 PL=0
MOVL C00432 V=800.0 PL=0
MOVL C00433 V=800.0 PL=0
MOVL C00434 V=800.0 PL=0
MOVL C00435 V=800.0 PL=0
MOVL C00436 V=800.0 PL=0
MOVL C00437 V=800.0 PL=0
MOVL C00438 V=800.0 PL=0
MOVL C00439 V=800.0 PL=0
MOVL C00440 V=800.0 PL=0
MOVL C00441 V=800.0 PL=0
MOVL C00442 V=800.0 PL=0
MOVL C00443 V=800.0 PL=0
MOVL C00444 V=800.0 PL=0
MOVL C00445 V=800.0 PL=0
MOVL C00446 V=800.0 PL=0
MOVL C00447 V=800.0 PL=0
MOVL C00448 V=800.0 PL=0
MOVL C00449 V=800.0 PL=0
MOVL C00450 V=800.0 PL=0
MOVL C00451 V=800.0 PL=0
MOVL C00452 V=800.0 PL=0
MOVL C00453 V=800.0 PL=0
MOVL C00454 V=800.0 PL=0
MOVL C00455 V=800.0 PL=0
MOVL C00456 V=800.0 PL=0
MOVL C00457 V=800.0 PL=0
MOVL C00458 V=800.0 PL=0
MOVL C00459 V=800.0 PL=0
MOVL C00460 V=800.0 PL=0
MOVL C00461 V=800.0 PL=0
MOVL C00462 V=800.0 PL=0
MOVL C00463 V=800.0 PL=0
MOVL C00464 V=800.0 PL=0
MOVL C00465 V=800.0 PL=0
MOVL C00466 V=800.0 PL=0
MOVL C00467 V=800.0 PL=0
MOVL C00468 V=800.0 PL=0
MOVL C00469 V=800.0 PL=0
MOVL C00470 V=800.0 PL=0
MOVL C00471 V=800.0 PL=0
MOVL C00472 V=800.0 PL=0
MOVL C00473 V=800.0 PL=0
MOVL C00474 V=800.0 PL=0
MOVL C00475 V=800.0 PL=0
MOVL C00476 V=800.0 PL=0
MOVL C00477 V=800.0 PL=0
MOVL C00478 V=800.0 PL=0
MOVL C00479 V=800.0 PL=0
MOVL C00480 V=800.0 PL=0
MOVL C00481 V=800.0 PL=0
MOVL C00482 V=800.0 PL=0
MOVL C00483 V=800.0 PL=0
MOVL C00484 V=800.0 PL=0
MOVL C00485 V=800.0 PL=0
MOVL C00486 V=800.0 PL=0
MOVL C00487 V=800.0 PL=0
MOVL C00488 V=800.0 PL=0
MOVL C00489 V=800.0 PL=0
MOVL C00490 V=800.0 PL=0
MOVL C00491 V=800.0 PL=0
MOVL C00492 V=800.0 PL=0
MOVL C00493 V=800.0 PL=0
MOVL C00494 V=800.0 PL=0
MOVL C00495 V=800.0 PL=0
MOVL C00496 V=800.0 PL=0
MOVL C00497 V=800.0 PL=0
MOVL C00498 V=800.0 PL=0
MOVL C00499 V=800.0 PL=0
MOVL C00500 V=800.0 PL=0
MOVL C00501 V=800.0 PL=0
MOVL C00502 V=800.0 PL=0
MOVL C00503 V=800.0 PL=0
MOVL C00504 V=800.0 PL=0
MOVL C00505 V=800.0 PL=0
MOVL C00506 V=800.0 PL=0
MOVL C00507 V=800.0 PL=0
MOVL C00508 V=800.0 PL=0
MOVL C00509 V=800.0 PL=0
MOVL C00510 V=800.0 PL=0
MOVL C00511 V=800.0 PL=0
MOVL C00512 V=800.0 PL=0
MOVL C00513 V=800.0 PL=0
MOVL C00514 V=800.0 PL=0
MOVL C00515 V=800.0 PL=0
MOVL C00516 V=800.0 PL=0
MOVL C00517 V=800.0 PL=0
MOVL C00518 V=800.0 PL=0
MOVL C00519 V=800.0 PL=0
MOVL C00520 V=800.0 PL=0
MOVL C00521 V=800.0 PL=0
MOVL C00522 V=800.0 PL=0
MOVL C00523 V=800.0 PL=0
MOVL C00524 V=800.0 PL=0
MOVL C00525 V=800.0 PL=0
MOVL C00526 V=800.0 PL=0
MOVL C00527 V=800.0 PL=0
MOVL C00528 V=800.0 PL=0
MOVL C00529 V=800.0 PL=0
MOVL C00530 V=800.0 PL=0
MOVL C00531 V=800.0 PL=0
MOVL C00532 V=800.0 PL=0
MOVL C00533 V=800.0 PL=0
MOVL C00534 V=800.0 PL=0
MOVL C00535 V=800.0 PL=0
MOVL C00536 V=800.0 PL=0
MOVL C00537 V=800.0 PL=0
MOVL C00538 V=800.0 PL=0
MOVL C00539 V=800.0 PL=0
MOVL C00540 V=800.0 PL=0
MOVL C00541 V=800.0 PL=0
MOVL C00542 V=800.0 PL=0
'CALL JOB: TOOL OFF
MOVJ C00543 VJ=25.00 PL=0
'CALL JOB: TOOL ON
MOVL C00544 V=800.0 PL=0
MOVL C00545 V=800.0 PL=0
MOVL C00546 V=800.0 PL=0
MOVL C00547 V=800.0 PL=0
MOVL C00548 V=800.0 PL=0
MOVL C00549 V=800.0 PL=0
MOVL C00550 V=800.0 PL=0
MOVL C00551 V=800.0 PL=0
MOVL C00552 V=800.0 PL=0
MOVL C00553 V=800.0 PL=0
MOVL C00554 V=800.0 PL=0
MOVL C00555 V=800.0 PL=0
MOVL C00556 V=800.0 PL=0
MOVL C00557 V=800.0 PL=0
MOVL C00558 V=800.0 PL=0
MOVL C00559 V=800.0 PL=0
MOVL C00560 V=800.0 PL=0
MOVL C00561 V=800.0 PL=0
MOVL C00562 V=800.0 PL=0
MOVL C00563 V=800.0 PL=0
MOVL C00564 V=800.0 PL=0
MOVL C00565 V=800.0 PL=0
'CALL JOB: TOOL OFF
MOVJ C00566 VJ=25.00 PL=0
'CALL JOB: TOOL ON
MOVL C00567 V=800.0 PL=0
MOVL C00568 V=800.0 PL=0
MOVL C00569 V=800.0 PL=0
MOVL C00570 V=800.0 PL=0
MOVL C00571 V=800.0 PL=0
MOVL C00572 V=800.0 PL=0
MOVL C00573 V=800.0 PL=0
MOVL C00574 V=800.0 PL=0
MOVL C00575 V=800.0 PL=0
MOVL C00576 V=800.0 PL=0
MOVL C00577 V=800.0 PL=0
MOVL C00578 V=800.0 PL=0
MOVL C00579 V=800.0 PL=0
MOVL C00580 V=800.0 PL=0
MOVL C00581 V=800.0 PL=0
MOVL C00582 V=800.0 PL=0
MOVL C00583 V=800.0 PL=0
MOVL C00584 V=800.0 PL=0
MOVL C00585 V=800.0 PL=0
MOVL C00586 V=800.0 PL=0
MOVL C00587 V=800.0 PL=0
MOVL C00588 V=800.0 PL=0
MOVL C00589 V=800.0 PL=0
MOVL C00590 V=800.0 PL=0
MOVL C00591 V=800.0 PL=0
MOVL C00592 V=800.0 PL=0
MOVL C00593 V=800.0 PL=0
MOVL C00594 V=800.0 PL=0
MOVL C00595 V=800.0 PL=0
MOVL C00596 V=800.0 PL=0
MOVL C00597 V=800.0 PL=0
MOVL C00598 V=800.0 PL=0
MOVL C00599 V=800.0 PL=0
MOVL C00600 V=800.0 PL=0
MOVL C00601 V=800.0 PL=0
MOVL C00602 V=800.0 PL=0
MOVL C00603 V=800.0 PL=0
MOVL C00604 V=800.0 PL=0
MOVL C00605 V=800.0 PL=0
MOVL C00606 V=800.0 PL=0
MOVL C00607 V=800.0 PL=0
MOVL C00608 V=800.0 PL=0
MOVL C00609 V=800.0 PL=0
MOVL C00610 V=800.0 PL=0
MOVL C00611 V=800.0 PL=0
MOVL C00612 V=800.0 PL=0
MOVL C00613 V=800.0 PL=0
MOVL C00614 V=800.0 PL=0
MOVL C00615 V=800.0 PL=0
MOVL C00616 V=800.0 PL=0
MOVL C00617 V=800.0 PL=0
MOVL C00618 V=800.0 PL=0
MOVL C00619 V=800.0 PL=0
MOVL C00620 V=800.0 PL=0
MOVL C00621 V=800.0 PL=0
MOVL C00622 V=800.0 PL=0
MOVL C00623 V=800.0 PL=0
MOVL C00624 V=800.0 PL=0
MOVL C00625 V=800.0 PL=0
MOVL C00626 V=800.0 PL=0
MOVL C00627 V=800.0 PL=0
MOVL C00628 V=800.0 PL=0
MOVL C00629 V=800.0 PL=0
MOVL C00630 V=800.0 PL=0
MOVL C00631 V=800.0 PL=0
MOVL C00632 V=800.0 PL=0
MOVL C00633 V=800.0 PL=0
MOVL C00634 V=800.0 PL=0
MOVL C00635 V=800.0 PL=0
MOVL C00636 V=800.0 PL=0
MOVL C00637 V=800.0 PL=0
MOVL C00638 V=800.0 PL=0
MOVL C00639 V=800.0 PL=0
MOVL C00640 V=800.0 PL=0
MOVL C00641 V=800.0 PL=0
MOVL C00642 V=800.0 PL=0
MOVL C00643 V=800.0 PL=0
MOVL C00644 V=800.0 PL=0
MOVL C00645 V=800.0 PL=0
MOVL C00646 V=800.0 PL=0
MOVL C00647 V=800.0 PL=0
MOVL C00648 V=800.0 PL=0
MOVL C00649 V=800.0 PL=0
MOVL C00650 V=800.0 PL=0
MOVL C00651 V=800.0 PL=0
MOVL C00652 V=800.0 PL=0
MOVL C00653 V=800.0 PL=0
MOVL C00654 V=800.0 PL=0
MOVL C00655 V=800.0 PL=0
MOVL C00656 V=800.0 PL=0
MOVL C00657 V=800.0 PL=0
MOVL C00658 V=800.0 PL=0
MOVL C00659 V=800.0 PL=0
MOVL C00660 V=800.0 PL=0
MOVL C00661 V=800.0 PL=0
MOVL C00662 V=800.0 PL=0
MOVL C00663 V=800.0 PL=0
MOVL C00664 V=800.0 PL=0
MOVL C00665 V=800.0 PL=0
MOVL C00666 V=800.0 PL=0
MOVL C00667 V=800.0 PL=0
MOVL C00668 V=800.0 PL=0
MOVL C00669 V=800.0 PL=0
MOVL C00670 V=800.0 PL=0
MOVL C00671 V=800.0 PL=0
MOVL C00672 V=800.0 PL=0
MOVL C00673 V=800.0 PL=0
MOVL C00674 V=800.0 PL=0
MOVL C00675 V=800.0 PL=0
MOVL C00676 V=800.0 PL=0
MOVL C00677 V=800.0 PL=0
MOVL C00678 V=800.0 PL=0
MOVL C00679 V=800.0 PL=0
MOVL C00680 V=800.0 PL=0
MOVL C00681 V=800.0 PL=0
MOVL C00682 V=800.0 PL=0
MOVL C00683 V=800.0 PL=0
MOVL C00684 V=800.0 PL=0
MOVL C00685 V=800.0 PL=0
MOVL C00686 V=800.0 PL=0
MOVL C00687 V=800.0 PL=0
MOVL C00688 V=800.0 PL=0
MOVL C00689 V=800.0 PL=0
MOVL C00690 V=800.0 PL=0
MOVL C00691 V=800.0 PL=0
MOVL C00692 V=800.0 PL=0
MOVL C00693 V=800.0 PL=0
MOVL C00694 V=800.0 PL=0
MOVL C00695 V=800.0 PL=0
MOVL C00696 V=800.0 PL=0
MOVL C00697 V=800.0 PL=0
MOVL C00698 V=800.0 PL=0
MOVL C00699 V=800.0 PL=0
MOVL C00700 V=800.0 PL=0
MOVL C00701 V=800.0 PL=0
MOVL C00702 V=800.0 PL=0
MOVL C00703 V=800.0 PL=0
MOVL C00704 V=800.0 PL=0
MOVL C00705 V=800.0 PL=0
MOVL C00706 V=800.0 PL=0
MOVL C00707 V=800.0 PL=0
MOVL C00708 V=800.0 PL=0
MOVL C00709 V=800.0 PL=0
MOVL C00710 V=800.0 PL=0
MOVL C00711 V=800.0 PL=0
MOVL C00712 V=800.0 PL=0
MOVL C00713 V=800.0 PL=0
MOVL C00714 V=800.0 PL=0
MOVL C00715 V=800.0 PL=0
MOVL C00716 V=800.0 PL=0
MOVL C00717 V=800.0 PL=0
MOVL C00718 V=800.0 PL=0
MOVL C00719 V=800.0 PL=0
MOVL C00720 V=800.0 PL=0
MOVL C00721 V=800.0 PL=0
MOVL C00722 V=800.0 PL=0
MOVL C00723 V=800.0 PL=0
MOVL C00724 V=800.0 PL=0
MOVL C00725 V=800.0 PL=0
MOVL C00726 V=800.0 PL=0
MOVL C00727 V=800.0 PL=0
MOVL C00728 V=800.0 PL=0
MOVL C00729 V=800.0 PL=0
MOVL C00730 V=800.0 PL=0
MOVL C00731 V=800.0 PL=0
MOVL C00732 V=800.0 PL=0
MOVL C00733 V=800.0 PL=0
MOVL C00734 V=800.0 PL=0
MOVL C00735 V=800.0 PL=0
MOVL C00736 V=800.0 PL=0
MOVL C00737 V=800.0 PL=0
MOVL C00738 V=800.0 PL=0
MOVL C00739 V=800.0 PL=0
MOVL C00740 V=800.0 PL=0
MOVL C00741 V=800.0 PL=0
MOVL C00742 V=800.0 PL=0
MOVL C00743 V=800.0 PL=0
MOVL C00744 V=800.0 PL=0
MOVL C00745 V=800.0 PL=0
MOVL C00746 V=800.0 PL=0
MOVL C00747 V=800.0 PL=0
MOVL C00748 V=800.0 PL=0
MOVL C00749 V=800.0 PL=0
MOVL C00750 V=800.0 PL=0
MOVL C00751 V=800.0 PL=0
MOVL C00752 V=800.0 PL=0
MOVL C00753 V=800.0 PL=0
MOVL C00754 V=800.0 PL=0
MOVL C00755 V=800.0 PL=0
MOVL C00756 V=800.0 PL=0
MOVL C00757 V=800.0 PL=0
MOVL C00758 V=800.0 PL=0
MOVL C00759 V=800.0 PL=0
MOVL C00760 V=800.0 PL=0
MOVL C00761 V=800.0 PL=0
MOVL C00762 V=800.0 PL=0
MOVL C00763 V=800.0 PL=0
MOVL C00764 V=800.0 PL=0
MOVL C00765 V=800.0 PL=0
MOVL C00766 V=800.0 PL=0
MOVL C00767 V=800.0 PL=0
MOVL C00768 V=800.0 PL=0
MOVL C00769 V=800.0 PL=0
MOVL C00770 V=800.0 PL=0
MOVL C00771 V=800.0 PL=0
MOVL C00772 V=800.0 PL=0
MOVL C00773 V=800.0 PL=0
MOVL C00774 V=800.0 PL=0
MOVL C00775 V=800.0 PL=0
MOVL C00776 V=800.0 PL=0
MOVL C00777 V=800.0 PL=0
MOVL C00778 V=800.0 PL=0
MOVL C00779 V=800.0 PL=0
MOVL C00780 V=800.0 PL=0
MOVL C00781 V=800.0 PL=0
MOVL C00782 V=800.0 PL=0
MOVL C00783 V=800.0 PL=0
MOVL C00784 V=800.0 PL=0
MOVL C00785 V=800.0 PL=0
MOVL C00786 V=800.0 PL=0
MOVL C00787 V=800.0 PL=0
MOVL C00788 V=800.0 PL=0
MOVL C00789 V=800.0 PL=0
MOVL C00790 V=800.0 PL=0
MOVL C00791 V=800.0 PL=0
MOVL C00792 V=800.0 PL=0
MOVL C00793 V=800.0 PL=0
MOVL C00794 V=800.0 PL=0
MOVL C00795 V=800.0 PL=0
MOVL C00796 V=800.0 PL=0
MOVL C00797 V=800.0 PL=0
MOVL C00798 V=800.0 PL=0
MOVL C00799 V=800.0 PL=0
MOVL C00800 V=800.0 PL=0
MOVL C00801 V=800.0 PL=0
MOVL C00802 V=800.0 PL=0
MOVL C00803 V=800.0 PL=0
MOVL C00804 V=800.0 PL=0
MOVL C00805 V=800.0 PL=0
MOVL C00806 V=800.0 PL=0
MOVL C00807 V=800.0 PL=0
MOVL C00808 V=800.0 PL=0
MOVL C00809 V=800.0 PL=0
MOVL C00810 V=800.0 PL=0
MOVL C00811 V=800.0 PL=0
MOVL C00812 V=800.0 PL=0
MOVL C00813 V=800.0 PL=0
MOVL C00814 V=800.0 PL=0
MOVL C00815 V=800.0 PL=0
MOVL C00816 V=800.0 PL=0
MOVL C00817 V=800.0 PL=0
MOVL C00818 V=800.0 PL=0
MOVL C00819 V=800.0 PL=0
MOVL C00820 V=800.0 PL=0
MOVL C00821 V=800.0 PL=0
MOVL C00822 V=800.0 PL=0
MOVL C00823 V=800.0 PL=0
MOVL C00824 V=800.0 PL=0
MOVL C00825 V=800.0 PL=0
MOVL C00826 V=800.0 PL=0
MOVL C00827 V=800.0 PL=0
MOVL C00828 V=800.0 PL=0
MOVL C00829 V=800.0 PL=0
MOVL C00830 V=800.0 PL=0
MOVL C00831 V=800.0 PL=0
MOVL C00832 V=800.0 PL=0
MOVL C00833 V=800.0 PL=0
MOVL C00834 V=800.0 PL=0
MOVL C00835 V=800.0 PL=0
MOVL C00836 V=800.0 PL=0
MOVL C00837 V=800.0 PL=0
MOVL C00838 V=800.0 PL=0
MOVL C00839 V=800.0 PL=0
MOVL C00840 V=800.0 PL=0
MOVL C00841 V=800.0 PL=0
MOVL C00842 V=800.0 PL=0
MOVL C00843 V=800.0 PL=0
MOVL C00844 V=800.0 PL=0
MOVL C00845 V=800.0 PL=0
MOVL C00846 V=800.0 PL=0
MOVL C00847 V=800.0 PL=0
MOVL C00848 V=800.0 PL=0
MOVL C00849 V=800.0 PL=0
MOVL C00850 V=800.0 PL=0
MOVL C00851 V=800.0 PL=0
MOVL C00852 V=800.0 PL=0
MOVL C00853 V=800.0 PL=0
MOVL C00854 V=800.0 PL=0
MOVL C00855 V=800.0 PL=0
MOVL C00856 V=800.0 PL=0
MOVL C00857 V=800.0 PL=0
MOVL C00858 V=800.0 PL=0
MOVL C00859 V=800.0 PL=0
MOVL C00860 V=800.0 PL=0
MOVL C00861 V=800.0 PL=0
MOVL C00862 V=800.0 PL=0
MOVL C00863 V=800.0 PL=0
MOVL C00864 V=800.0 PL=0
MOVL C00865 V=800.0 PL=0
MOVL C00866 V=800.0 PL=0
MOVL C00867 V=800.0 PL=0
MOVL C00868 V=800.0 PL=0
MOVL C00869 V=800.0 PL=0
MOVL C00870 V=800.0 PL=0
MOVL C00871 V=800.0 PL=0
MOVL C00872 V=800.0 PL=0
MOVL C00873 V=800.0 PL=0
MOVL C00874 V=800.0 PL=0
MOVL C00875 V=800.0 PL=0
MOVL C00876 V=800.0 PL=0
MOVL C00877 V=800.0 PL=0
MOVL C00878 V=800.0 PL=0
MOVL C00879 V=800.0 PL=0
MOVL C00880 V=800.0 PL=0
MOVL C00881 V=800.0 PL=0
MOVL C00882 V=800.0 PL=0
MOVL C00883 V=800.0 PL=0
MOVL C00884 V=800.0 PL=0
MOVL C00885 V=800.0 PL=0
MOVL C00886 V=800.0 PL=0
MOVL C00887 V=800.0 PL=0
MOVL C00888 V=800.0 PL=0
MOVL C00889 V=800.0 PL=0
MOVL C00890 V=800.0 PL=0
MOVL C00891 V=800.0 PL=0
MOVL C00892 V=800.0 PL=0
MOVL C00893 V=800.0 PL=0
MOVL C00894 V=800.0 PL=0
MOVL C00895 V=800.0 PL=0
MOVL C00896 V=800.0 PL=0
MOVL C00897 V=800.0 PL=0
MOVL C00898 V=800.0 PL=0
MOVL C00899 V=800.0 PL=0
MOVL C00900 V=800.0 PL=0
MOVL C00901 V=800.0 PL=0
MOVL C00902 V=800.0 PL=0
MOVL C00903 V=800.0 PL=0
MOVL C00904 V=800.0 PL=0
MOVL C00905 V=800.0 PL=0
MOVL C00906 V=800.0 PL=0
MOVL C00907 V=800.0 PL=0
MOVL C00908 V=800.0 PL=0
MOVL C00909 V=800.0 PL=0
MOVL C00910 V=800.0 PL=0
MOVL C00911 V=800.0 PL=0
MOVL C00912 V=800.0 PL=0
MOVL C00913 V=800.0 PL=0
MOVL C00914 V=800.0 PL=0
MOVL C00915 V=800.0 PL=0
MOVL C00916 V=800.0 PL=0
MOVL C00917 V=800.0 PL=0
MOVL C00918 V=800.0 PL=0
MOVL C00919 V=800.0 PL=0
MOVL C00920 V=800.0 PL=0
MOVL C00921 V=800.0 PL=0
MOVL C00922 V=800.0 PL=0
MOVL C00923 V=800.0 PL=0
MOVL C00924 V=800.0 PL=0
MOVL C00925 V=800.0 PL=0
MOVL C00926 V=800.0 PL=0
MOVL C00927 V=800.0 PL=0
MOVL C00928 V=800.0 PL=0
MOVL C00929 V=800.0 PL=0
MOVL C00930 V=800.0 PL=0
MOVL C00931 V=800.0 PL=0
MOVL C00932 V=800.0 PL=0
MOVL C00933 V=800.0 PL=0
MOVL C00934 V=800.0 PL=0
MOVL C00935 V=800.0 PL=0
MOVL C00936 V=800.0 PL=0
MOVL C00937 V=800.0 PL=0
MOVL C00938 V=800.0 PL=0
MOVL C00939 V=800.0 PL=0
MOVL C00940 V=800.0 PL=0
MOVL C00941 V=800.0 PL=0
MOVL C00942 V=800.0 PL=0
MOVL C00943 V=800.0 PL=0
MOVL C00944 V=800.0 PL=0
MOVL C00945 V=800.0 PL=0
MOVL C00946 V=800.0 PL=0
MOVL C00947 V=800.0 PL=0
MOVL C00948 V=800.0 PL=0
MOVL C00949 V=800.0 PL=0
MOVL C00950 V=800.0 PL=0
MOVL C00951 V=800.0 PL=0
MOVL C00952 V=800.0 PL=0
MOVL C00953 V=800.0 PL=0
MOVL C00954 V=800.0 PL=0
MOVL C00955 V=800.0 PL=0
MOVL C00956 V=800.0 PL=0
MOVL C00957 V=800.0 PL=0
MOVL C00958 V=800.0 PL=0
MOVL C00959 V=800.0 PL=0
MOVL C00960 V=800.0 PL=0
MOVL C00961 V=800.0 PL=0
MOVL C00962 V=800.0 PL=0
MOVL C00963 V=800.0 PL=0
MOVL C00964 V=800.0 PL=0
MOVL C00965 V=800.0 PL=0
MOVL C00966 V=800.0 PL=0
MOVL C00967 V=800.0 PL=0
MOVL C00968 V=800.0 PL=0
MOVL C00969 V=800.0 PL=0
MOVL C00970 V=800.0 PL=0
MOVL C00971 V=800.0 PL=0
'CALL JOB: TOOL OFF
MOVJ C00972 VJ=25.00 PL=0
'CALL JOB: TOOL ON
MOVL C00973 V=800.0 PL=0
MOVL C00974 V=800.0 PL=0
MOVL C00975 V=800.0 PL=0
MOVL C00976 V=800.0 PL=0
MOVL C00977 V=800.0 PL=0
MOVL C00978 V=800.0 PL=0
MOVL C00979 V=800.0 PL=0
MOVL C00980 V=800.0 PL=0
MOVL C00981 V=800.0 PL=0
MOVL C00982 V=800.0 PL=0
MOVL C00983 V=800.0 PL=0
MOVL C00984 V=800.0 PL=0
MOVL C00985 V=800.0 PL=0
MOVL C00986 V=800.0 PL=0
MOVL C00987 V=800.0 PL=0
MOVL C00988 V=800.0 PL=0
MOVL C00989 V=800.0 PL=0
MOVL C00990 V=800.0 PL=0
MOVL C00991 V=800.0 PL=0
MOVL C00992 V=800.0 PL=0
MOVL C00993 V=800.0 PL=0
MOVL C00994 V=800.0 PL=0
MOVL C00995 V=800.0 PL=0
MOVL C00996 V=800.0 PL=0
MOVL C00997 V=800.0 PL=0
MOVL C00998 V=800.0 PL=0
MOVL C00999 V=800.0 PL=0
MOVL C01000 V=800.0 PL=0
MOVL C01001 V=800.0 PL=0
MOVL C01002 V=800.0 PL=0
MOVL C01003 V=800.0 PL=0
MOVL C01004 V=800.0 PL=0
MOVL C01005 V=800.0 PL=0
MOVL C01006 V=800.0 PL=0
MOVL C01007 V=800.0 PL=0
MOVL C01008 V=800.0 PL=0
MOVL C01009 V=800.0 PL=0
MOVL C01010 V=800.0 PL=0
MOVL C01011 V=800.0 PL=0
MOVL C01012 V=800.0 PL=0
MOVL C01013 V=800.0 PL=0
MOVL C01014 V=800.0 PL=0
MOVL C01015 V=800.0 PL=0
MOVL C01016 V=800.0 PL=0
MOVL C01017 V=800.0 PL=0
MOVL C01018 V=800.0 PL=0
MOVL C01019 V=800.0 PL=0
MOVL C01020 V=800.0 PL=0
MOVL C01021 V=800.0 PL=0
MOVL C01022 V=800.0 PL=0
MOVL C01023 V=800.0 PL=0
MOVL C01024 V=800.0 PL=0
MOVL C01025 V=800.0 PL=0
MOVL C01026 V=800.0 PL=0
MOVL C01027 V=800.0 PL=0
MOVL C01028 V=800.0 PL=0
MOVL C01029 V=800.0 PL=0
MOVL C01030 V=800.0 PL=0
MOVL C01031 V=800.0 PL=0
MOVL C01032 V=800.0 PL=0
MOVL C01033 V=800.0 PL=0
MOVL C01034 V=800.0 PL=0
MOVL C01035 V=800.0 PL=0
MOVL C01036 V=800.0 PL=0
MOVL C01037 V=800.0 PL=0
MOVL C01038 V=800.0 PL=0
MOVL C01039 V=800.0 PL=0
MOVL C01040 V=800.0 PL=0
MOVL C01041 V=800.0 PL=0
MOVL C01042 V=800.0 PL=0
MOVL C01043 V=800.0 PL=0
MOVL C01044 V=800.0 PL=0
MOVL C01045 V=800.0 PL=0
MOVL C01046 V=800.0 PL=0
MOVL C01047 V=800.0 PL=0
MOVL C01048 V=800.0 PL=0
MOVL C01049 V=800.0 PL=0
MOVL C01050 V=800.0 PL=0
MOVL C01051 V=800.0 PL=0
MOVL C01052 V=800.0 PL=0
MOVL C01053 V=800.0 PL=0
MOVL C01054 V=800.0 PL=0
MOVL C01055 V=800.0 PL=0
MOVL C01056 V=800.0 PL=0
MOVL C01057 V=800.0 PL=0
MOVL C01058 V=800.0 PL=0
MOVL C01059 V=800.0 PL=0
MOVL C01060 V=800.0 PL=0
MOVL C01061 V=800.0 PL=0
MOVL C01062 V=800.0 PL=0
MOVL C01063 V=800.0 PL=0
MOVL C01064 V=800.0 PL=0
MOVL C01065 V=800.0 PL=0
MOVL C01066 V=800.0 PL=0
MOVL C01067 V=800.0 PL=0
MOVL C01068 V=800.0 PL=0
MOVL C01069 V=800.0 PL=0
MOVL C01070 V=800.0 PL=0
MOVL C01071 V=800.0 PL=0
MOVL C01072 V=800.0 PL=0
MOVL C01073 V=800.0 PL=0
MOVL C01074 V=800.0 PL=0
MOVL C01075 V=800.0 PL=0
MOVL C01076 V=800.0 PL=0
MOVL C01077 V=800.0 PL=0
MOVL C01078 V=800.0 PL=0
MOVL C01079 V=800.0 PL=0
MOVL C01080 V=800.0 PL=0
MOVL C01081 V=800.0 PL=0
MOVL C01082 V=800.0 PL=0
MOVL C01083 V=800.0 PL=0
MOVL C01084 V=800.0 PL=0
MOVL C01085 V=800.0 PL=0
MOVL C01086 V=800.0 PL=0
MOVL C01087 V=800.0 PL=0
MOVL C01088 V=800.0 PL=0
MOVL C01089 V=800.0 PL=0
MOVL C01090 V=800.0 PL=0
MOVL C01091 V=800.0 PL=0
MOVL C01092 V=800.0 PL=0
MOVL C01093 V=800.0 PL=0
MOVL C01094 V=800.0 PL=0
MOVL C01095 V=800.0 PL=0
MOVL C01096 V=800.0 PL=0
MOVL C01097 V=800.0 PL=0
MOVL C01098 V=800.0 PL=0
MOVL C01099 V=800.0 PL=0
MOVL C01100 V=800.0 PL=0
MOVL C01101 V=800.0 PL=0
MOVL C01102 V=800.0 PL=0
MOVL C01103 V=800.0 PL=0
MOVL C01104 V=800.0 PL=0
MOVL C01105 V=800.0 PL=0
MOVL C01106 V=800.0 PL=0
MOVL C01107 V=800.0 PL=0
MOVL C01108 V=800.0 PL=0
MOVL C01109 V=800.0 PL=0
MOVL C01110 V=800.0 PL=0
MOVL C01111 V=800.0 PL=0
MOVL C01112 V=800.0 PL=0
MOVL C01113 V=800.0 PL=0
MOVL C01114 V=800.0 PL=0
MOVL C01115 V=800.0 PL=0
MOVL C01116 V=800.0 PL=0
MOVL C01117 V=800.0 PL=0
MOVL C01118 V=800.0 PL=0
MOVL C01119 V=800.0 PL=0
MOVL C01120 V=800.0 PL=0
MOVL C01121 V=800.0 PL=0
MOVL C01122 V=800.0 PL=0
MOVL C01123 V=800.0 PL=0
MOVL C01124 V=800.0 PL=0
MOVL C01125 V=800.0 PL=0
MOVL C01126 V=800.0 PL=0
MOVL C01127 V=800.0 PL=0
MOVL C01128 V=800.0 PL=0
MOVL C01129 V=800.0 PL=0
MOVL C01130 V=800.0 PL=0
MOVL C01131 V=800.0 PL=0
MOVL C01132 V=800.0 PL=0
MOVL C01133 V=800.0 PL=0
MOVL C01134 V=800.0 PL=0
MOVL C01135 V=800.0 PL=0
MOVL C01136 V=800.0 PL=0
MOVL C01137 V=800.0 PL=0
MOVL C01138 V=800.0 PL=0
MOVL C01139 V=800.0 PL=0
MOVL C01140 V=800.0 PL=0
MOVL C01141 V=800.0 PL=0
MOVL C01142 V=800.0 PL=0
MOVL C01143 V=800.0 PL=0
MOVL C01144 V=800.0 PL=0
MOVL C01145 V=800.0 PL=0
MOVL C01146 V=800.0 PL=0
MOVL C01147 V=800.0 PL=0
MOVL C01148 V=800.0 PL=0
MOVL C01149 V=800.0 PL=0
MOVL C01150 V=800.0 PL=0
MOVL C01151 V=800.0 PL=0
MOVL C01152 V=800.0 PL=0
MOVL C01153 V=800.0 PL=0
MOVL C01154 V=800.0 PL=0
MOVL C01155 V=800.0 PL=0
MOVL C01156 V=800.0 PL=0
MOVL C01157 V=800.0 PL=0
MOVL C01158 V=800.0 PL=0
MOVL C01159 V=800.0 PL=0
MOVL C01160 V=800.0 PL=0
MOVL C01161 V=800.0 PL=0
MOVL C01162 V=800.0 PL=0
MOVL C01163 V=800.0 PL=0
MOVL C01164 V=800.0 PL=0
MOVL C01165 V=800.0 PL=0
MOVL C01166 V=800.0 PL=0
MOVL C01167 V=800.0 PL=0
MOVL C01168 V=800.0 PL=0
MOVL C01169 V=800.0 PL=0
MOVL C01170 V=800.0 PL=0
MOVL C01171 V=800.0 PL=0
MOVL C01172 V=800.0 PL=0
MOVL C01173 V=800.0 PL=0
MOVL C01174 V=800.0 PL=0
MOVL C01175 V=800.0 PL=0
MOVL C01176 V=800.0 PL=0
MOVL C01177 V=800.0 PL=0
MOVL C01178 V=800.0 PL=0
MOVL C01179 V=800.0 PL=0
MOVL C01180 V=800.0 PL=0
MOVL C01181 V=800.0 PL=0
MOVL C01182 V=800.0 PL=0
MOVL C01183 V=800.0 PL=0
MOVL C01184 V=800.0 PL=0
MOVL C01185 V=800.0 PL=0
MOVL C01186 V=800.0 PL=0
MOVL C01187 V=800.0 PL=0
MOVL C01188 V=800.0 PL=0
MOVL C01189 V=800.0 PL=0
MOVL C01190 V=800.0 PL=0
MOVL C01191 V=800.0 PL=0
MOVL C01192 V=800.0 PL=0
MOVL C01193 V=800.0 PL=0
MOVL C01194 V=800.0 PL=0
MOVL C01195 V=800.0 PL=0
MOVL C01196 V=800.0 PL=0
MOVL C01197 V=800.0 PL=0
MOVL C01198 V=800.0 PL=0
MOVL C01199 V=800.0 PL=0
MOVL C01200 V=800.0 PL=0
MOVL C01201 V=800.0 PL=0
MOVL C01202 V=800.0 PL=0
MOVL C01203 V=800.0 PL=0
MOVL C01204 V=800.0 PL=0
MOVL C01205 V=800.0 PL=0
MOVL C01206 V=800.0 PL=0
MOVL C01207 V=800.0 PL=0
MOVL C01208 V=800.0 PL=0
MOVL C01209 V=800.0 PL=0
MOVL C01210 V=800.0 PL=0
MOVL C01211 V=800.0 PL=0
MOVL C01212 V=800.0 PL=0
MOVL C01213 V=800.0 PL=0
MOVL C01214 V=800.0 PL=0
MOVL C01215 V=800.0 PL=0
MOVL C01216 V=800.0 PL=0
MOVL C01217 V=800.0 PL=0
MOVL C01218 V=800.0 PL=0
MOVL C01219 V=800.0 PL=0
MOVL C01220 V=800.0 PL=0
MOVL C01221 V=800.0 PL=0
MOVL C01222 V=800.0 PL=0
MOVL C01223 V=800.0 PL=0
MOVL C01224 V=800.0 PL=0
MOVL C01225 V=800.0 PL=0
MOVL C01226 V=800.0 PL=0
MOVL C01227 V=800.0 PL=0
MOVL C01228 V=800.0 PL=0
MOVL C01229 V=800.0 PL=0
MOVL C01230 V=800.0 PL=0
MOVL C01231 V=800.0 PL=0
MOVL C01232 V=800.0 PL=0
MOVL C01233 V=800.0 PL=0
MOVL C01234 V=800.0 PL=0
MOVL C01235 V=800.0 PL=0
MOVL C01236 V=800.0 PL=0
MOVL C01237 V=800.0 PL=0
MOVL C01238 V=800.0 PL=0
MOVL C01239 V=800.0 PL=0
MOVL C01240 V=800.0 PL=0
MOVL C01241 V=800.0 PL=0
MOVL C01242 V=800.0 PL=0
MOVL C01243 V=800.0 PL=0
MOVL C01244 V=800.0 PL=0
MOVL C01245 V=800.0 PL=0
MOVL C01246 V=800.0 PL=0
MOVL C01247 V=800.0 PL=0
MOVL C01248 V=800.0 PL=0
MOVL C01249 V=800.0 PL=0
MOVL C01250 V=800.0 PL=0
MOVL C01251 V=800.0 PL=0
MOVL C01252 V=800.0 PL=0
MOVL C01253 V=800.0 PL=0
MOVL C01254 V=800.0 PL=0
MOVL C01255 V=800.0 PL=0
MOVL C01256 V=800.0 PL=0
MOVL C01257 V=800.0 PL=0
MOVL C01258 V=800.0 PL=0
MOVL C01259 V=800.0 PL=0
MOVL C01260 V=800.0 PL=0
MOVL C01261 V=800.0 PL=0
MOVL C01262 V=800.0 PL=0
MOVL C01263 V=800.0 PL=0
MOVL C01264 V=800.0 PL=0
MOVL C01265 V=800.0 PL=0
MOVL C01266 V=800.0 PL=0
MOVL C01267 V=800.0 PL=0
MOVL C01268 V=800.0 PL=0
MOVL C01269 V=800.0 PL=0
MOVL C01270 V=800.0 PL=0
MOVL C01271 V=800.0 PL=0
MOVL C01272 V=800.0 PL=0
MOVL C01273 V=800.0 PL=0
MOVL C01274 V=800.0 PL=0
MOVL C01275 V=800.0 PL=0
MOVL C01276 V=800.0 PL=0
MOVL C01277 V=800.0 PL=0
MOVL C01278 V=800.0 PL=0
MOVL C01279 V=800.0 PL=0
MOVL C01280 V=800.0 PL=0
MOVL C01281 V=800.0 PL=0
MOVL C01282 V=800.0 PL=0
MOVL C01283 V=800.0 PL=0
MOVL C01284 V=800.0 PL=0
MOVL C01285 V=800.0 PL=0
MOVL C01286 V=800.0 PL=0
MOVL C01287 V=800.0 PL=0
MOVL C01288 V=800.0 PL=0
MOVL C01289 V=800.0 PL=0
MOVL C01290 V=800.0 PL=0
MOVL C01291 V=800.0 PL=0
MOVL C01292 V=800.0 PL=0
MOVL C01293 V=800.0 PL=0
MOVL C01294 V=800.0 PL=0
MOVL C01295 V=800.0 PL=0
MOVL C01296 V=800.0 PL=0
MOVL C01297 V=800.0 PL=0
MOVL C01298 V=800.0 PL=0
MOVL C01299 V=800.0 PL=0
MOVL C01300 V=800.0 PL=0
MOVL C01301 V=800.0 PL=0
MOVL C01302 V=800.0 PL=0
MOVL C01303 V=800.0 PL=0
MOVL C01304 V=800.0 PL=0
MOVL C01305 V=800.0 PL=0
MOVL C01306 V=800.0 PL=0
MOVL C01307 V=800.0 PL=0
MOVL C01308 V=800.0 PL=0
MOVL C01309 V=800.0 PL=0
MOVL C01310 V=800.0 PL=0
MOVL C01311 V=800.0 PL=0
MOVL C01312 V=800.0 PL=0
MOVL C01313 V=800.0 PL=0
MOVL C01314 V=800.0 PL=0
MOVL C01315 V=800.0 PL=0
MOVL C01316 V=800.0 PL=0
MOVL C01317 V=800.0 PL=0
MOVL C01318 V=800.0 PL=0
MOVL C01319 V=800.0 PL=0
MOVL C01320 V=800.0 PL=0
MOVL C01321 V=800.0 PL=0
MOVL C01322 V=800.0 PL=0
MOVL C01323 V=800.0 PL=0
MOVL C01324 V=800.0 PL=0
MOVL C01325 V=800.0 PL=0
MOVL C01326 V=800.0 PL=0
MOVL C01327 V=800.0 PL=0
MOVL C01328 V=800.0 PL=0
MOVL C01329 V=800.0 PL=0
MOVL C01330 V=800.0 PL=0
MOVL C01331 V=800.0 PL=0
MOVL C01332 V=800.0 PL=0
MOVL C01333 V=800.0 PL=0
MOVL C01334 V=800.0 PL=0
MOVL C01335 V=800.0 PL=0
MOVL C01336 V=800.0 PL=0
MOVL C01337 V=800.0 PL=0
MOVL C01338 V=800.0 PL=0
MOVL C01339 V=800.0 PL=0
MOVL C01340 V=800.0 PL=0
MOVL C01341 V=800.0 PL=0
MOVL C01342 V=800.0 PL=0
MOVL C01343 V=800.0 PL=0
MOVL C01344 V=800.0 PL=0
MOVL C01345 V=800.0 PL=0
MOVL C01346 V=800.0 PL=0
MOVL C01347 V=800.0 PL=0
MOVL C01348 V=800.0 PL=0
MOVL C01349 V=800.0 PL=0
MOVL C01350 V=800.0 PL=0
MOVL C01351 V=800.0 PL=0
MOVL C01352 V=800.0 PL=0
MOVL C01353 V=800.0 PL=0
MOVL C01354 V=800.0 PL=0
MOVL C01355 V=800.0 PL=0
MOVL C01356 V=800.0 PL=0
MOVL C01357 V=800.0 PL=0
MOVL C01358 V=800.0 PL=0
MOVL C01359 V=800.0 PL=0
MOVL C01360 V=800.0 PL=0
MOVL C01361 V=800.0 PL=0
MOVL C01362 V=800.0 PL=0
MOVL C01363 V=800.0 PL=0
MOVL C01364 V=800.0 PL=0
MOVL C01365 V=800.0 PL=0
MOVL C01366 V=800.0 PL=0
MOVL C01367 V=800.0 PL=0
MOVL C01368 V=800.0 PL=0
MOVL C01369 V=800.0 PL=0
MOVL C01370 V=800.0 PL=0
MOVL C01371 V=800.0 PL=0
MOVL C01372 V=800.0 PL=0
MOVL C01373 V=800.0 PL=0
MOVL C01374 V=800.0 PL=0
MOVL C01375 V=800.0 PL=0
MOVL C01376 V=800.0 PL=0
MOVL C01377 V=800.0 PL=0
MOVL C01378 V=800.0 PL=0
MOVL C01379 V=800.0 PL=0
MOVL C01380 V=800.0 PL=0
MOVL C01381 V=800.0 PL=0
MOVL C01382 V=800.0 PL=0
MOVL C01383 V=800.0 PL=0
MOVL C01384 V=800.0 PL=0
MOVL C01385 V=800.0 PL=0
MOVL C01386 V=800.0 PL=0
MOVL C01387 V=800.0 PL=0
MOVL C01388 V=800.0 PL=0
MOVL C01389 V=800.0 PL=0
MOVL C01390 V=800.0 PL=0
MOVL C01391 V=800.0 PL=0
MOVL C01392 V=800.0 PL=0
MOVL C01393 V=800.0 PL=0
MOVL C01394 V=800.0 PL=0
MOVL C01395 V=800.0 PL=0
MOVL C01396 V=800.0 PL=0
MOVL C01397 V=800.0 PL=0
MOVL C01398 V=800.0 PL=0
MOVL C01399 V=800.0 PL=0
MOVL C01400 V=800.0 PL=0
MOVL C01401 V=800.0 PL=0
MOVL C01402 V=800.0 PL=0
MOVL C01403 V=800.0 PL=0
MOVL C01404 V=800.0 PL=0
MOVL C01405 V=800.0 PL=0
MOVL C01406 V=800.0 PL=0
MOVL C01407 V=800.0 PL=0
MOVL C01408 V=800.0 PL=0
MOVL C01409 V=800.0 PL=0
MOVL C01410 V=800.0 PL=0
MOVL C01411 V=800.0 PL=0
MOVL C01412 V=800.0 PL=0
MOVL C01413 V=800.0 PL=0
MOVL C01414 V=800.0 PL=0
MOVL C01415 V=800.0 PL=0
MOVL C01416 V=800.0 PL=0
MOVL C01417 V=800.0 PL=0
MOVL C01418 V=800.0 PL=0
MOVL C01419 V=800.0 PL=0
MOVL C01420 V=800.0 PL=0
MOVL C01421 V=800.0 PL=0
MOVL C01422 V=800.0 PL=0
MOVL C01423 V=800.0 PL=0
MOVL C01424 V=800.0 PL=0
MOVL C01425 V=800.0 PL=0
MOVL C01426 V=800.0 PL=0
MOVL C01427 V=800.0 PL=0
MOVL C01428 V=800.0 PL=0
MOVL C01429 V=800.0 PL=0
MOVL C01430 V=800.0 PL=0
MOVL C01431 V=800.0 PL=0
MOVL C01432 V=800.0 PL=0
MOVL C01433 V=800.0 PL=0
MOVL C01434 V=800.0 PL=0
MOVL C01435 V=800.0 PL=0
MOVL C01436 V=800.0 PL=0
MOVL C01437 V=800.0 PL=0
MOVL C01438 V=800.0 PL=0
MOVL C01439 V=800.0 PL=0
MOVL C01440 V=800.0 PL=0
MOVL C01441 V=800.0 PL=0
MOVL C01442 V=800.0 PL=0
MOVL C01443 V=800.0 PL=0
MOVL C01444 V=800.0 PL=0
MOVL C01445 V=800.0 PL=0
MOVL C01446 V=800.0 PL=0
MOVL C01447 V=800.0 PL=0
MOVL C01448 V=800.0 PL=0
MOVL C01449 V=800.0 PL=0
MOVL C01450 V=800.0 PL=0
MOVL C01451 V=800.0 PL=0
MOVL C01452 V=800.0 PL=0
MOVL C01453 V=800.0 PL=0
MOVL C01454 V=800.0 PL=0
MOVL C01455 V=800.0 PL=0
MOVL C01456 V=800.0 PL=0
MOVL C01457 V=800.0 PL=0
MOVL C01458 V=800.0 PL=0
MOVL C01459 V=800.0 PL=0
MOVL C01460 V=800.0 PL=0
MOVL C01461 V=800.0 PL=0
MOVL C01462 V=800.0 PL=0
MOVL C01463 V=800.0 PL=0
MOVL C01464 V=800.0 PL=0
MOVL C01465 V=800.0 PL=0
MOVL C01466 V=800.0 PL=0
MOVL C01467 V=800.0 PL=0
MOVL C01468 V=800.0 PL=0
MOVL C01469 V=800.0 PL=0
MOVL C01470 V=800.0 PL=0
MOVL C01471 V=800.0 PL=0
MOVL C01472 V=800.0 PL=0
MOVL C01473 V=800.0 PL=0
MOVL C01474 V=800.0 PL=0
MOVL C01475 V=800.0 PL=0
MOVL C01476 V=800.0 PL=0
MOVL C01477 V=800.0 PL=0
MOVL C01478 V=800.0 PL=0
MOVL C01479 V=800.0 PL=0
MOVL C01480 V=800.0 PL=0
MOVL C01481 V=800.0 PL=0
MOVL C01482 V=800.0 PL=0
MOVL C01483 V=800.0 PL=0
MOVL C01484 V=800.0 PL=0
MOVL C01485 V=800.0 PL=0
MOVL C01486 V=800.0 PL=0
MOVL C01487 V=800.0 PL=0
MOVL C01488 V=800.0 PL=0
MOVL C01489 V=800.0 PL=0
MOVL C01490 V=800.0 PL=0
MOVL C01491 V=800.0 PL=0
MOVL C01492 V=800.0 PL=0
MOVL C01493 V=800.0 PL=0
MOVL C01494 V=800.0 PL=0
MOVL C01495 V=800.0 PL=0
MOVL C01496 V=800.0 PL=0
MOVL C01497 V=800.0 PL=0
MOVL C01498 V=800.0 PL=0
MOVL C01499 V=800.0 PL=0
MOVL C01500 V=800.0 PL=0
MOVL C01501 V=800.0 PL=0
MOVL C01502 V=800.0 PL=0
MOVL C01503 V=800.0 PL=0
MOVL C01504 V=800.0 PL=0
MOVL C01505 V=800.0 PL=0
MOVL C01506 V=800.0 PL=0
MOVL C01507 V=800.0 PL=0
MOVL C01508 V=800.0 PL=0
MOVL C01509 V=800.0 PL=0
MOVL C01510 V=800.0 PL=0
MOVL C01511 V=800.0 PL=0
MOVL C01512 V=800.0 PL=0
MOVL C01513 V=800.0 PL=0
MOVL C01514 V=800.0 PL=0
MOVL C01515 V=800.0 PL=0
MOVL C01516 V=800.0 PL=0
MOVL C01517 V=800.0 PL=0
MOVL C01518 V=800.0 PL=0
MOVL C01519 V=800.0 PL=0
MOVL C01520 V=800.0 PL=0
MOVL C01521 V=800.0 PL=0
MOVL C01522 V=800.0 PL=0
MOVL C01523 V=800.0 PL=0
MOVL C01524 V=800.0 PL=0
MOVL C01525 V=800.0 PL=0
MOVL C01526 V=800.0 PL=0
MOVL C01527 V=800.0 PL=0
MOVL C01528 V=800.0 PL=0
MOVL C01529 V=800.0 PL=0
MOVL C01530 V=800.0 PL=0
MOVL C01531 V=800.0 PL=0
MOVL C01532 V=800.0 PL=0
MOVL C01533 V=800.0 PL=0
MOVL C01534 V=800.0 PL=0
MOVL C01535 V=800.0 PL=0
MOVL C01536 V=800.0 PL=0
MOVL C01537 V=800.0 PL=0
MOVL C01538 V=800.0 PL=0
MOVL C01539 V=800.0 PL=0
MOVL C01540 V=800.0 PL=0
MOVL C01541 V=800.0 PL=0
MOVL C01542 V=800.0 PL=0
MOVL C01543 V=800.0 PL=0
MOVL C01544 V=800.0 PL=0
MOVL C01545 V=800.0 PL=0
MOVL C01546 V=800.0 PL=0
MOVL C01547 V=800.0 PL=0
MOVL C01548 V=800.0 PL=0
MOVL C01549 V=800.0 PL=0
MOVL C01550 V=800.0 PL=0
MOVL C01551 V=800.0 PL=0
MOVL C01552 V=800.0 PL=0
MOVL C01553 V=800.0 PL=0
MOVL C01554 V=800.0 PL=0
MOVL C01555 V=800.0 PL=0
MOVL C01556 V=800.0 PL=0
MOVL C01557 V=800.0 PL=0
MOVL C01558 V=800.0 PL=0
MOVL C01559 V=800.0 PL=0
MOVL C01560 V=800.0 PL=0
MOVL C01561 V=800.0 PL=0
MOVL C01562 V=800.0 PL=0
MOVL C01563 V=800.0 PL=0
MOVL C01564 V=800.0 PL=0
MOVL C01565 V=800.0 PL=0
MOVL C01566 V=800.0 PL=0
MOVL C01567 V=800.0 PL=0
MOVL C01568 V=800.0 PL=0
MOVL C01569 V=800.0 PL=0
MOVL C01570 V=800.0 PL=0
MOVL C01571 V=800.0 PL=0
MOVL C01572 V=800.0 PL=0
MOVL C01573 V=800.0 PL=0
MOVL C01574 V=800.0 PL=0
MOVL C01575 V=800.0 PL=0
MOVL C01576 V=800.0 PL=0
MOVL C01577 V=800.0 PL=0
MOVL C01578 V=800.0 PL=0
MOVL C01579 V=800.0 PL=0
MOVL C01580 V=800.0 PL=0
MOVL C01581 V=800.0 PL=0
MOVL C01582 V=800.0 PL=0
MOVL C01583 V=800.0 PL=0
MOVL C01584 V=800.0 PL=0
MOVL C01585 V=800.0 PL=0
MOVL C01586 V=800.0 PL=0
MOVL C01587 V=800.0 PL=0
MOVL C01588 V=800.0 PL=0
MOVL C01589 V=800.0 PL=0
MOVL C01590 V=800.0 PL=0
MOVL C01591 V=800.0 PL=0
MOVL C01592 V=800.0 PL=0
MOVL C01593 V=800.0 PL=0
MOVL C01594 V=800.0 PL=0
MOVL C01595 V=800.0 PL=0
MOVL C01596 V=800.0 PL=0
MOVL C01597 V=800.0 PL=0
MOVL C01598 V=800.0 PL=0
MOVL C01599 V=800.0 PL=0
MOVL C01600 V=800.0 PL=0
MOVL C01601 V=800.0 PL=0
MOVL C01602 V=800.0 PL=0
MOVL C01603 V=800.0 PL=0
MOVL C01604 V=800.0 PL=0
MOVL C01605 V=800.0 PL=0
MOVL C01606 V=800.0 PL=0
MOVL C01607 V=800.0 PL=0
MOVL C01608 V=800.0 PL=0
MOVL C01609 V=800.0 PL=0
MOVL C01610 V=800.0 PL=0
MOVL C01611 V=800.0 PL=0
MOVL C01612 V=800.0 PL=0
MOVL C01613 V=800.0 PL=0
MOVL C01614 V=800.0 PL=0
MOVL C01615 V=800.0 PL=0
MOVL C01616 V=800.0 PL=0
MOVL C01617 V=800.0 PL=0
MOVL C01618 V=800.0 PL=0
MOVL C01619 V=800.0 PL=0
MOVL C01620 V=800.0 PL=0
MOVL C01621 V=800.0 PL=0
MOVL C01622 V=800.0 PL=0
MOVL C01623 V=800.0 PL=0
MOVL C01624 V=800.0 PL=0
MOVL C01625 V=800.0 PL=0
MOVL C01626 V=800.0 PL=0
MOVL C01627 V=800.0 PL=0
MOVL C01628 V=800.0 PL=0
MOVL C01629 V=800.0 PL=0
MOVL C01630 V=800.0 PL=0
MOVL C01631 V=800.0 PL=0
MOVL C01632 V=800.0 PL=0
MOVL C01633 V=800.0 PL=0
MOVL C01634 V=800.0 PL=0
MOVL C01635 V=800.0 PL=0
MOVL C01636 V=800.0 PL=0
MOVL C01637 V=800.0 PL=0
MOVL C01638 V=800.0 PL=0
MOVL C01639 V=800.0 PL=0
MOVL C01640 V=800.0 PL=0
MOVL C01641 V=800.0 PL=0
MOVL C01642 V=800.0 PL=0
MOVL C01643 V=800.0 PL=0
MOVL C01644 V=800.0 PL=0
MOVL C01645 V=800.0 PL=0
MOVL C01646 V=800.0 PL=0
MOVL C01647 V=800.0 PL=0
MOVL C01648 V=800.0 PL=0
MOVL C01649 V=800.0 PL=0
MOVL C01650 V=800.0 PL=0
MOVL C01651 V=800.0 PL=0
MOVL C01652 V=800.0 PL=0
MOVL C01653 V=800.0 PL=0
MOVL C01654 V=800.0 PL=0
MOVL C01655 V=800.0 PL=0
MOVL C01656 V=800.0 PL=0
MOVL C01657 V=800.0 PL=0
MOVL C01658 V=800.0 PL=0
MOVL C01659 V=800.0 PL=0
MOVL C01660 V=800.0 PL=0
MOVL C01661 V=800.0 PL=0
MOVL C01662 V=800.0 PL=0
MOVL C01663 V=800.0 PL=0
MOVL C01664 V=800.0 PL=0
MOVL C01665 V=800.0 PL=0
MOVL C01666 V=800.0 PL=0
MOVL C01667 V=800.0 PL=0
MOVL C01668 V=800.0 PL=0
MOVL C01669 V=800.0 PL=0
MOVL C01670 V=800.0 PL=0
MOVL C01671 V=800.0 PL=0
MOVL C01672 V=800.0 PL=0
MOVL C01673 V=800.0 PL=0
MOVL C01674 V=800.0 PL=0
MOVL C01675 V=800.0 PL=0
MOVL C01676 V=800.0 PL=0
MOVL C01677 V=800.0 PL=0
MOVL C01678 V=800.0 PL=0
MOVL C01679 V=800.0 PL=0
MOVL C01680 V=800.0 PL=0
MOVL C01681 V=800.0 PL=0
MOVL C01682 V=800.0 PL=0
MOVL C01683 V=800.0 PL=0
MOVL C01684 V=800.0 PL=0
MOVL C01685 V=800.0 PL=0
MOVL C01686 V=800.0 PL=0
MOVL C01687 V=800.0 PL=0
MOVL C01688 V=800.0 PL=0
MOVL C01689 V=800.0 PL=0
MOVL C01690 V=800.0 PL=0
MOVL C01691 V=800.0 PL=0
MOVL C01692 V=800.0 PL=0
MOVL C01693 V=800.0 PL=0
MOVL C01694 V=800.0 PL=0
MOVL C01695 V=800.0 PL=0
MOVL C01696 V=800.0 PL=0
MOVL C01697 V=800.0 PL=0
MOVL C01698 V=800.0 PL=0
MOVL C01699 V=800.0 PL=0
MOVL C01700 V=800.0 PL=0
MOVL C01701 V=800.0 PL=0
MOVL C01702 V=800.0 PL=0
MOVL C01703 V=800.0 PL=0
MOVL C01704 V=800.0 PL=0
MOVL C01705 V=800.0 PL=0
MOVL C01706 V=800.0 PL=0
MOVL C01707 V=800.0 PL=0
MOVL C01708 V=800.0 PL=0
MOVL C01709 V=800.0 PL=0
MOVL C01710 V=800.0 PL=0
MOVL C01711 V=800.0 PL=0
MOVL C01712 V=800.0 PL=0
MOVL C01713 V=800.0 PL=0
MOVL C01714 V=800.0 PL=0
MOVL C01715 V=800.0 PL=0
MOVL C01716 V=800.0 PL=0
MOVL C01717 V=800.0 PL=0
MOVL C01718 V=800.0 PL=0
MOVL C01719 V=800.0 PL=0
MOVL C01720 V=800.0 PL=0
MOVL C01721 V=800.0 PL=0
MOVL C01722 V=800.0 PL=0
MOVL C01723 V=800.0 PL=0
MOVL C01724 V=800.0 PL=0
MOVL C01725 V=800.0 PL=0
MOVL C01726 V=800.0 PL=0
MOVL C01727 V=800.0 PL=0
MOVL C01728 V=800.0 PL=0
MOVL C01729 V=800.0 PL=0
MOVL C01730 V=800.0 PL=0
MOVL C01731 V=800.0 PL=0
MOVL C01732 V=800.0 PL=0
MOVL C01733 V=800.0 PL=0
MOVL C01734 V=800.0 PL=0
MOVL C01735 V=800.0 PL=0
MOVL C01736 V=800.0 PL=0
MOVL C01737 V=800.0 PL=0
MOVL C01738 V=800.0 PL=0
MOVL C01739 V=800.0 PL=0
MOVL C01740 V=800.0 PL=0
MOVL C01741 V=800.0 PL=0
MOVL C01742 V=800.0 PL=0
MOVL C01743 V=800.0 PL=0
MOVL C01744 V=800.0 PL=0
MOVL C01745 V=800.0 PL=0
MOVL C01746 V=800.0 PL=0
MOVL C01747 V=800.0 PL=0
MOVL C01748 V=800.0 PL=0
MOVL C01749 V=800.0 PL=0
MOVL C01750 V=800.0 PL=0
MOVL C01751 V=800.0 PL=0
MOVL C01752 V=800.0 PL=0
MOVL C01753 V=800.0 PL=0
MOVL C01754 V=800.0 PL=0
MOVL C01755 V=800.0 PL=0
MOVL C01756 V=800.0 PL=0
MOVL C01757 V=800.0 PL=0
MOVL C01758 V=800.0 PL=0
MOVL C01759 V=800.0 PL=0
MOVL C01760 V=800.0 PL=0
MOVL C01761 V=800.0 PL=0
MOVL C01762 V=800.0 PL=0
MOVL C01763 V=800.0 PL=0
MOVL C01764 V=800.0 PL=0
MOVL C01765 V=800.0 PL=0
MOVL C01766 V=800.0 PL=0
MOVL C01767 V=800.0 PL=0
MOVL C01768 V=800.0 PL=0
MOVL C01769 V=800.0 PL=0
MOVL C01770 V=800.0 PL=0
MOVL C01771 V=800.0 PL=0
MOVL C01772 V=800.0 PL=0
MOVL C01773 V=800.0 PL=0
MOVL C01774 V=800.0 PL=0
MOVL C01775 V=800.0 PL=0
MOVL C01776 V=800.0 PL=0
MOVL C01777 V=800.0 PL=0
MOVL C01778 V=800.0 PL=0
MOVL C01779 V=800.0 PL=0
MOVL C01780 V=800.0 PL=0
MOVL C01781 V=800.0 PL=0
MOVL C01782 V=800.0 PL=0
MOVL C01783 V=800.0 PL=0
MOVL C01784 V=800.0 PL=0
MOVL C01785 V=800.0 PL=0
MOVL C01786 V=800.0 PL=0
MOVL C01787 V=800.0 PL=0
MOVL C01788 V=800.0 PL=0
MOVL C01789 V=800.0 PL=0
MOVL C01790 V=800.0 PL=0
MOVL C01791 V=800.0 PL=0
MOVL C01792 V=800.0 PL=0
MOVL C01793 V=800.0 PL=0
MOVL C01794 V=800.0 PL=0
MOVL C01795 V=800.0 PL=0
MOVL C01796 V=800.0 PL=0
MOVL C01797 V=800.0 PL=0
MOVL C01798 V=800.0 PL=0
MOVL C01799 V=800.0 PL=0
MOVL C01800 V=800.0 PL=0
MOVL C01801 V=800.0 PL=0
MOVL C01802 V=800.0 PL=0
MOVL C01803 V=800.0 PL=0
MOVL C01804 V=800.0 PL=0
MOVL C01805 V=800.0 PL=0
MOVL C01806 V=800.0 PL=0
MOVL C01807 V=800.0 PL=0
MOVL C01808 V=800.0 PL=0
MOVL C01809 V=800.0 PL=0
MOVL C01810 V=800.0 PL=0
MOVL C01811 V=800.0 PL=0
MOVL C01812 V=800.0 PL=0
MOVL C01813 V=800.0 PL=0
MOVL C01814 V=800.0 PL=0
MOVL C01815 V=800.0 PL=0
MOVL C01816 V=800.0 PL=0
MOVL C01817 V=800.0 PL=0
MOVL C01818 V=800.0 PL=0
MOVL C01819 V=800.0 PL=0
MOVL C01820 V=800.0 PL=0
MOVL C01821 V=800.0 PL=0
MOVL C01822 V=800.0 PL=0
MOVL C01823 V=800.0 PL=0
MOVL C01824 V=800.0 PL=0
MOVL C01825 V=800.0 PL=0
MOVL C01826 V=800.0 PL=0
MOVL C01827 V=800.0 PL=0
MOVL C01828 V=800.0 PL=0
MOVL C01829 V=800.0 PL=0
MOVL C01830 V=800.0 PL=0
MOVL C01831 V=800.0 PL=0
MOVL C01832 V=800.0 PL=0
MOVL C01833 V=800.0 PL=0
MOVL C01834 V=800.0 PL=0
MOVL C01835 V=800.0 PL=0
MOVL C01836 V=800.0 PL=0
MOVL C01837 V=800.0 PL=0
MOVL C01838 V=800.0 PL=0
MOVL C01839 V=800.0 PL=0
MOVL C01840 V=800.0 PL=0
MOVL C01841 V=800.0 PL=0
MOVL C01842 V=800.0 PL=0
MOVL C01843 V=800.0 PL=0
MOVL C01844 V=800.0 PL=0
MOVL C01845 V=800.0 PL=0
MOVL C01846 V=800.0 PL=0
MOVL C01847 V=800.0 PL=0
MOVL C01848 V=800.0 PL=0
MOVL C01849 V=800.0 PL=0
MOVL C01850 V=800.0 PL=0
MOVL C01851 V=800.0 PL=0
MOVL C01852 V=800.0 PL=0
MOVL C01853 V=800.0 PL=0
MOVL C01854 V=800.0 PL=0
MOVL C01855 V=800.0 PL=0
MOVL C01856 V=800.0 PL=0
MOVL C01857 V=800.0 PL=0
MOVL C01858 V=800.0 PL=0
MOVL C01859 V=800.0 PL=0
MOVL C01860 V=800.0 PL=0
MOVL C01861 V=800.0 PL=0
MOVL C01862 V=800.0 PL=0
MOVL C01863 V=800.0 PL=0
MOVL C01864 V=800.0 PL=0
MOVL C01865 V=800.0 PL=0
MOVL C01866 V=800.0 PL=0
MOVL C01867 V=800.0 PL=0
MOVL C01868 V=800.0 PL=0
MOVL C01869 V=800.0 PL=0
MOVL C01870 V=800.0 PL=0
MOVL C01871 V=800.0 PL=0
MOVL C01872 V=800.0 PL=0
MOVL C01873 V=800.0 PL=0
MOVL C01874 V=800.0 PL=0
MOVL C01875 V=800.0 PL=0
MOVL C01876 V=800.0 PL=0
MOVL C01877 V=800.0 PL=0
MOVL C01878 V=800.0 PL=0
MOVL C01879 V=800.0 PL=0
MOVL C01880 V=800.0 PL=0
MOVL C01881 V=800.0 PL=0
MOVL C01882 V=800.0 PL=0
MOVL C01883 V=800.0 PL=0
MOVL C01884 V=800.0 PL=0
MOVL C01885 V=800.0 PL=0
MOVL C01886 V=800.0 PL=0
MOVL C01887 V=800.0 PL=0
MOVL C01888 V=800.0 PL=0
MOVL C01889 V=800.0 PL=0
MOVL C01890 V=800.0 PL=0
MOVL C01891 V=800.0 PL=0
MOVL C01892 V=800.0 PL=0
MOVL C01893 V=800.0 PL=0
MOVL C01894 V=800.0 PL=0
MOVL C01895 V=800.0 PL=0
MOVL C01896 V=800.0 PL=0
MOVL C01897 V=800.0 PL=0
MOVL C01898 V=800.0 PL=0
MOVL C01899 V=800.0 PL=0
MOVL C01900 V=800.0 PL=0
MOVL C01901 V=800.0 PL=0
MOVL C01902 V=800.0 PL=0
MOVL C01903 V=800.0 PL=0
MOVL C01904 V=800.0 PL=0
MOVL C01905 V=800.0 PL=0
MOVL C01906 V=800.0 PL=0
MOVL C01907 V=800.0 PL=0
MOVL C01908 V=800.0 PL=0
MOVL C01909 V=800.0 PL=0
MOVL C01910 V=800.0 PL=0
MOVL C01911 V=800.0 PL=0
MOVL C01912 V=800.0 PL=0
MOVL C01913 V=800.0 PL=0
MOVL C01914 V=800.0 PL=0
MOVL C01915 V=800.0 PL=0
MOVL C01916 V=800.0 PL=0
MOVL C01917 V=800.0 PL=0
MOVL C01918 V=800.0 PL=0
MOVL C01919 V=800.0 PL=0
MOVL C01920 V=800.0 PL=0
MOVL C01921 V=800.0 PL=0
MOVL C01922 V=800.0 PL=0
MOVL C01923 V=800.0 PL=0
MOVL C01924 V=800.0 PL=0
MOVL C01925 V=800.0 PL=0
MOVL C01926 V=800.0 PL=0
MOVL C01927 V=800.0 PL=0
MOVL C01928 V=800.0 PL=0
MOVL C01929 V=800.0 PL=0
MOVL C01930 V=800.0 PL=0
MOVL C01931 V=800.0 PL=0
MOVL C01932 V=800.0 PL=0
MOVL C01933 V=800.0 PL=0
MOVL C01934 V=800.0 PL=0
MOVL C01935 V=800.0 PL=0
MOVL C01936 V=800.0 PL=0
MOVL C01937 V=800.0 PL=0
MOVL C01938 V=800.0 PL=0
MOVL C01939 V=800.0 PL=0
MOVL C01940 V=800.0 PL=0
MOVL C01941 V=800.0 PL=0
MOVL C01942 V=800.0 PL=0
MOVL C01943 V=800.0 PL=0
MOVL C01944 V=800.0 PL=0
MOVL C01945 V=800.0 PL=0
MOVL C01946 V=800.0 PL=0
MOVL C01947 V=800.0 PL=0
MOVL C01948 V=800.0 PL=0
MOVL C01949 V=800.0 PL=0
MOVL C01950 V=800.0 PL=0
MOVL C01951 V=800.0 PL=0
MOVL C01952 V=800.0 PL=0
MOVL C01953 V=800.0 PL=0
MOVL C01954 V=800.0 PL=0
MOVL C01955 V=800.0 PL=0
MOVL C01956 V=800.0 PL=0
MOVL C01957 V=800.0 PL=0
MOVL C01958 V=800.0 PL=0
MOVL C01959 V=800.0 PL=0
MOVL C01960 V=800.0 PL=0
MOVL C01961 V=800.0 PL=0
MOVL C01962 V=800.0 PL=0
MOVL C01963 V=800.0 PL=0
MOVL C01964 V=800.0 PL=0
MOVL C01965 V=800.0 PL=0
MOVL C01966 V=800.0 PL=0
MOVL C01967 V=800.0 PL=0
MOVL C01968 V=800.0 PL=0
MOVL C01969 V=800.0 PL=0
MOVL C01970 V=800.0 PL=0
MOVL C01971 V=800.0 PL=0
MOVL C01972 V=800.0 PL=0
MOVL C01973 V=800.0 PL=0
MOVL C01974 V=800.0 PL=0
MOVL C01975 V=800.0 PL=0
MOVL C01976 V=800.0 PL=0
MOVL C01977 V=800.0 PL=0
MOVL C01978 V=800.0 PL=0
MOVL C01979 V=800.0 PL=0
MOVL C01980 V=800.0 PL=0
MOVL C01981 V=800.0 PL=0
MOVL C01982 V=800.0 PL=0
MOVL C01983 V=800.0 PL=0
MOVL C01984 V=800.0 PL=0
MOVL C01985 V=800.0 PL=0
MOVL C01986 V=800.0 PL=0
MOVL C01987 V=800.0 PL=0
MOVL C01988 V=800.0 PL=0
MOVL C01989 V=800.0 PL=0
MOVL C01990 V=800.0 PL=0
MOVL C01991 V=800.0 PL=0
MOVL C01992 V=800.0 PL=0
MOVL C01993 V=800.0 PL=0
MOVL C01994 V=800.0 PL=0
MOVL C01995 V=800.0 PL=0
MOVL C01996 V=800.0 PL=0
MOVL C01997 V=800.0 PL=0
MOVL C01998 V=800.0 PL=0
MOVL C01999 V=800.0 PL=0
MOVL C02000 V=800.0 PL=0
MOVL C02001 V=800.0 PL=0
MOVL C02002 V=800.0 PL=0
MOVL C02003 V=800.0 PL=0
MOVL C02004 V=800.0 PL=0
MOVL C02005 V=800.0 PL=0
MOVL C02006 V=800.0 PL=0
MOVL C02007 V=800.0 PL=0
MOVL C02008 V=800.0 PL=0
MOVL C02009 V=800.0 PL=0
MOVL C02010 V=800.0 PL=0
MOVL C02011 V=800.0 PL=0
MOVL C02012 V=800.0 PL=0
MOVL C02013 V=800.0 PL=0
MOVL C02014 V=800.0 PL=0
MOVL C02015 V=800.0 PL=0
MOVL C02016 V=800.0 PL=0
MOVL C02017 V=800.0 PL=0
MOVL C02018 V=800.0 PL=0
MOVL C02019 V=800.0 PL=0
MOVL C02020 V=800.0 PL=0
MOVL C02021 V=800.0 PL=0
MOVL C02022 V=800.0 PL=0
MOVL C02023 V=800.0 PL=0
MOVL C02024 V=800.0 PL=0
MOVL C02025 V=800.0 PL=0
MOVL C02026 V=800.0 PL=0
MOVL C02027 V=800.0 PL=0
MOVL C02028 V=800.0 PL=0
MOVL C02029 V=800.0 PL=0
MOVL C02030 V=800.0 PL=0
MOVL C02031 V=800.0 PL=0
MOVL C02032 V=800.0 PL=0
MOVL C02033 V=800.0 PL=0
MOVL C02034 V=800.0 PL=0
MOVL C02035 V=800.0 PL=0
MOVL C02036 V=800.0 PL=0
MOVL C02037 V=800.0 PL=0
MOVL C02038 V=800.0 PL=0
MOVL C02039 V=800.0 PL=0
MOVL C02040 V=800.0 PL=0
MOVL C02041 V=800.0 PL=0
MOVL C02042 V=800.0 PL=0
MOVL C02043 V=800.0 PL=0
MOVL C02044 V=800.0 PL=0
MOVL C02045 V=800.0 PL=0
MOVL C02046 V=800.0 PL=0
MOVL C02047 V=800.0 PL=0
MOVL C02048 V=800.0 PL=0
MOVL C02049 V=800.0 PL=0
MOVL C02050 V=800.0 PL=0
MOVL C02051 V=800.0 PL=0
MOVL C02052 V=800.0 PL=0
MOVL C02053 V=800.0 PL=0
MOVL C02054 V=800.0 PL=0
MOVL C02055 V=800.0 PL=0
MOVL C02056 V=800.0 PL=0
MOVL C02057 V=800.0 PL=0
MOVL C02058 V=800.0 PL=0
MOVL C02059 V=800.0 PL=0
MOVL C02060 V=800.0 PL=0
MOVL C02061 V=800.0 PL=0
MOVL C02062 V=800.0 PL=0
MOVL C02063 V=800.0 PL=0
MOVL C02064 V=800.0 PL=0
MOVL C02065 V=800.0 PL=0
MOVL C02066 V=800.0 PL=0
MOVL C02067 V=800.0 PL=0
MOVL C02068 V=800.0 PL=0
MOVL C02069 V=800.0 PL=0
MOVL C02070 V=800.0 PL=0
MOVL C02071 V=800.0 PL=0
MOVL C02072 V=800.0 PL=0
MOVL C02073 V=800.0 PL=0
MOVL C02074 V=800.0 PL=0
MOVL C02075 V=800.0 PL=0
MOVL C02076 V=800.0 PL=0
MOVL C02077 V=800.0 PL=0
MOVL C02078 V=800.0 PL=0
MOVL C02079 V=800.0 PL=0
